(* Logix 5000 project; controller reports 1756-L63 rev 20.15; software revision 20.04; part 44 of 52 *)

        [122].log_data[40].maxminute := 25, [122].log_data[40].valid := 1, [122].log_data[41].min := 0.022540038, [122].log_data[41].max := 0.023128908, [122].log_data[41].total := 82.19256, [122].log_data[41].time := 3600.0, [122].log_data[41].minminute := 6, [122].log_data[41].maxminute := 1, [122].log_data[41].valid := 1, [122].log_data[42].min := 2.2911716, [122].log_data[42].max := 2.2963536, [122].log_data[42].total := 8258.403, [122].log_data[42].time := 3600.0, [122].log_data[42].minminute := 22, [122].log_data[42].maxminute := 41, [122].log_data[42].valid := 1, [122].log_data[43].min := -0.27999878, [122].log_data[43].max := -0.26000214, [122].log_data[43].total := -936.05817, [122].log_data[43].time := 3600.0, [122].log_data[43].minminute := 7, [122].log_data[43].valid := 1, [122].log_data[44].min := -0.30000305, [122].log_data[44].max := -0.27999878, [122].log_data[44].total := -1080.0862, [122].log_data[44].time := 3600.0, [122].log_data[44].maxminute := 20, [122].log_data[44].valid := 1, [122].log_data[45].time := 3600.0, [122].log_data[45].valid := 1, [122].log_data[46].time := 3600.0, [122].log_data[46].valid := 1, [122].log_data[47].time := 3600.0, [122].log_data[47].valid := 1, [122].log_data[48].min := 6.554947, [122].log_data[48].max := 6.9405026, [122].log_data[48].total := 24061.553, [122].log_data[48].time := 3600.0, [122].log_data[48].minminute := 51, [122].log_data[48].maxminute := 30, [122].log_data[48].valid := 1, [122].log_data[49].min := 9.374254, [122].log_data[49].max := 9.504003, [122].log_data[49].total := 34030.01, [122].log_data[49].time := 3600.0, [122].log_data[49].minminute := 59, [122].log_data[49].maxminute := 15, [122].log_data[49].valid := 1, [122].log_data[50].min := 1.5897048, [122].log_data[50].max := 1.6947598, [122].log_data[50].total := 5915.742, [122].log_data[50].time := 3600.0, [122].log_data[50].minminute := 30, [122].log_data[50].maxminute := 37, [122].log_data[50].valid := 1, [122].log_data[51].time := 3600.0, [122].log_data[51].valid := 1, [122].log_data[52].min := -2.959999, [122].log_data[52].max := 0.11999512, [122].log_data[52].total := -7874.2905,
        [122].log_data[52].time := 3600.0, [122].log_data[52].minminute := 54, [122].log_data[52].valid := 1, [122].log_data[53].min := -2.5800018, [122].log_data[53].max := 0.13999939, [122].log_data[53].total := -7446.6367, [122].log_data[53].time := 3600.0, [122].log_data[53].minminute := 9, [122].log_data[53].maxminute := 7, [122].log_data[53].valid := 1, [122].log_data[54].max := 0.5335, [122].log_data[54].total := 1217.6704, [122].log_data[54].time := 3600.0, [122].log_data[54].maxminute := 54, [122].log_data[54].valid := 1, [122].log_data[55].max := 0.5115, [122].log_data[55].total := 1217.3799, [122].log_data[55].time := 3600.0, [122].log_data[55].minminute := 5, [122].log_data[55].maxminute := 7, [122].log_data[55].valid := 1, [122].log_data[56].min := 0.15926416, [122].log_data[56].max := 0.159696, [122].log_data[56].total := 573.94727, [122].log_data[56].time := 3600.0, [122].log_data[56].minminute := 33, [122].log_data[56].maxminute := 2, [122].log_data[56].valid := 1, [122].log_data[57].min := 0.21273394, [122].log_data[57].max := 0.21501088, [122].log_data[57].total := 772.2598, [122].log_data[57].time := 3600.0, [122].log_data[57].minminute := 59, [122].log_data[57].maxminute := 6, [122].log_data[57].valid := 1, [122].log_data[58].time := 3600.0, [122].log_data[58].valid := 1, [122].log_data[59].time := 3600.0, [122].log_data[59].valid := 1, [122].log_data[60].valid := 1, [122].log_data[61].valid := 1, [122].log_data[62].valid := 1, [122].log_data[63].valid := 1, [122].log_data[64].valid := 1, [122].log_data[65].valid := 1, [122].log_data[66].valid := 1, [122].log_data[67].valid := 1, [122].log_data[68].valid := 1, [122].log_data[69].valid := 1, [122].log_data[70].valid := 1, [122].log_data[71].valid := 1, [122].log_data[72].valid := 1, [122].log_data[73].valid := 1, [122].log_data[74].valid := 1, [122].log_data[75].valid := 1, [122].log_data[76].valid := 1, [122].log_data[77].valid := 1, [122].log_data[78].valid := 1, [122].log_data[79].valid := 1, [122].log_data[80].valid := 1,
        [122].log_data[81].valid := 1, [122].log_data[82].valid := 1, [122].log_data[83].valid := 1, [122].log_data[84].valid := 1, [122].log_data[85].valid := 1, [122].log_data[86].valid := 1, [122].log_data[87].valid := 1, [122].log_data[88].valid := 1, [122].log_data[89].valid := 1, [122].log_data[90].valid := 1, [122].log_data[91].valid := 1, [122].log_data[92].valid := 1, [122].log_data[93].valid := 1, [122].log_data[94].valid := 1, [122].log_data[95].valid := 1, [122].log_data[96].valid := 1, [122].log_data[97].valid := 1, [122].log_data[98].valid := 1, [122].log_data[99].valid := 1, [122].log_data[100].valid := 1, [122].log_data[101].valid := 1, [122].log_data[102].valid := 1, [122].log_data[103].valid := 1, [122].log_data[104].valid := 1, [122].log_data[105].valid := 1, [122].log_data[106].valid := 1, [122].log_data[107].valid := 1, [122].log_data[108].valid := 1, [122].log_data[109].valid := 1, [122].log_data[110].valid := 1, [122].log_data[111].valid := 1, [122].log_data[112].valid := 1, [122].log_data[113].valid := 1, [122].log_data[114].valid := 1, [122].log_data[115].valid := 1, [122].log_data[116].valid := 1, [122].log_data[117].valid := 1, [122].log_data[118].valid := 1, [122].log_data[119].valid := 1, [122].log_data[120].valid := 1, [122].log_data[121].valid := 1, [122].log_data[122].valid := 1, [122].log_data[123].valid := 1, [122].log_data[124].valid := 1, [122].time.Year := 2023, [122].time.Month := 1, [122].time.Day := 18, [122].time.Hour := 5, [122].time.Minute := 59, [122].time.Second := 59, [123].log_data[0].min := 1.0, [123].log_data[0].max := 1.0, [123].log_data[0].total := 3600.0, [123].log_data[0].time := 3600.0, [123].log_data[0].valid := 1, [123].log_data[1].time := 3600.0, [123].log_data[1].valid := 1, [123].log_data[2].time := 3600.0, [123].log_data[2].valid := 1, [123].log_data[3].time := 3600.0,
        [123].log_data[3].valid := 1, [123].log_data[4].time := 3600.0, [123].log_data[4].valid := 1, [123].log_data[5].time := 3600.0, [123].log_data[5].valid := 1, [123].log_data[6].time := 3600.0, [123].log_data[6].valid := 1, [123].log_data[7].time := 3600.0, [123].log_data[7].valid := 1, [123].log_data[8].min := 1.0, [123].log_data[8].max := 1.0, [123].log_data[8].total := 3600.0, [123].log_data[8].time := 3600.0, [123].log_data[8].valid := 1, [123].log_data[9].min := 1.0, [123].log_data[9].max := 1.0, [123].log_data[9].total := 3600.0, [123].log_data[9].time := 3600.0, [123].log_data[9].valid := 1, [123].log_data[10].min := 1.0, [123].log_data[10].max := 1.0, [123].log_data[10].total := 3600.0, [123].log_data[10].time := 3600.0, [123].log_data[10].valid := 1, [123].log_data[11].time := 3600.0, [123].log_data[11].valid := 1, [123].log_data[12].min := 1.0, [123].log_data[12].max := 1.0, [123].log_data[12].total := 3600.0, [123].log_data[12].time := 3600.0, [123].log_data[12].valid := 1, [123].log_data[13].min := 1.0, [123].log_data[13].max := 1.0, [123].log_data[13].total := 3600.0, [123].log_data[13].time := 3600.0, [123].log_data[13].valid := 1, [123].log_data[14].time := 3600.0, [123].log_data[14].valid := 1, [123].log_data[15].time := 3600.0, [123].log_data[15].valid := 1, [123].log_data[16].time := 3600.0, [123].log_data[16].valid := 1, [123].log_data[17].min := 1.0, [123].log_data[17].max := 1.0, [123].log_data[17].total := 3600.0, [123].log_data[17].time := 3600.0, [123].log_data[17].valid := 1, [123].log_data[18].time := 3600.0, [123].log_data[18].valid := 1, [123].log_data[19].time := 3600.0, [123].log_data[19].valid := 1, [123].log_data[20].time := 3600.0, [123].log_data[20].valid := 1, [123].log_data[21].min := 1.0, [123].log_data[21].max := 1.0, [123].log_data[21].total := 3600.0, [123].log_data[21].time := 3600.0, [123].log_data[21].valid := 1, [123].log_data[22].time := 3600.0, [123].log_data[22].valid := 1,
        [123].log_data[23].time := 3600.0, [123].log_data[23].valid := 1, [123].log_data[24].time := 3600.0, [123].log_data[24].valid := 1, [123].log_data[25].time := 3600.0, [123].log_data[25].valid := 1, [123].log_data[26].time := 3600.0, [123].log_data[26].valid := 1, [123].log_data[27].time := 3600.0, [123].log_data[27].valid := 1, [123].log_data[28].time := 3600.0, [123].log_data[28].valid := 1, [123].log_data[29].min := 1.0, [123].log_data[29].max := 1.0, [123].log_data[29].total := 3600.0, [123].log_data[29].time := 3600.0, [123].log_data[29].valid := 1, [123].log_data[30].min := 1.0, [123].log_data[30].max := 1.0, [123].log_data[30].total := 3600.0, [123].log_data[30].time := 3600.0, [123].log_data[30].valid := 1, [123].log_data[31].max := 1.0, [123].log_data[31].total := 1440.998, [123].log_data[31].time := 3600.0, [123].log_data[31].minminute := 3, [123].log_data[31].valid := 1, [123].log_data[32].max := 1.0, [123].log_data[32].total := 1630.249, [123].log_data[32].time := 3600.0, [123].log_data[32].maxminute := 4, [123].log_data[32].valid := 1, [123].log_data[33].time := 3600.0, [123].log_data[33].valid := 1, [123].log_data[34].time := 3600.0, [123].log_data[34].valid := 1, [123].log_data[35].max := 1.0, [123].log_data[35].total := 1549.2471, [123].log_data[35].time := 3600.0, [123].log_data[35].maxminute := 10, [123].log_data[35].valid := 1, [123].log_data[36].max := 1.0, [123].log_data[36].total := 1609.498, [123].log_data[36].time := 3600.0, [123].log_data[36].minminute := 8, [123].log_data[36].valid := 1, [123].log_data[37].time := 3600.0, [123].log_data[37].valid := 1, [123].log_data[38].time := 3600.0, [123].log_data[38].valid := 1, [123].log_data[39].min := 0.9947063, [123].log_data[39].max := 1.0056593, [123].log_data[39].total := 3606.119, [123].log_data[39].time := 3600.0, [123].log_data[39].minminute := 20, [123].log_data[39].maxminute := 17, [123].log_data[39].valid := 1, [123].log_data[40].min := 7.602789, [123].log_data[40].max := 7.609111, [123].log_data[40].total := 27387.07,
        [123].log_data[40].time := 3600.0, [123].log_data[40].minminute := 1, [123].log_data[40].valid := 1, [123].log_data[41].min := 0.022540038, [123].log_data[41].max := 0.023128908, [123].log_data[41].total := 82.054955, [123].log_data[41].time := 3600.0, [123].log_data[41].maxminute := 55, [123].log_data[41].valid := 1, [123].log_data[42].min := 2.2912893, [123].log_data[42].max := 2.296118, [123].log_data[42].total := 8258.289, [123].log_data[42].time := 3600.0, [123].log_data[42].minminute := 33, [123].log_data[42].maxminute := 34, [123].log_data[42].valid := 1, [123].log_data[43].min := -0.27999878, [123].log_data[43].max := -0.26000214, [123].log_data[43].total := -936.1481, [123].log_data[43].time := 3600.0, [123].log_data[43].minminute := 14, [123].log_data[43].valid := 1, [123].log_data[44].min := -0.30000305, [123].log_data[44].max := -0.27999878, [123].log_data[44].total := -1080.081, [123].log_data[44].time := 3600.0, [123].log_data[44].valid := 1, [123].log_data[45].time := 3600.0, [123].log_data[45].valid := 1, [123].log_data[46].time := 3600.0, [123].log_data[46].valid := 1, [123].log_data[47].time := 3600.0, [123].log_data[47].valid := 1, [123].log_data[48].min := 6.64371, [123].log_data[48].max := 6.799526, [123].log_data[48].total := 24267.373, [123].log_data[48].time := 3600.0, [123].log_data[48].maxminute := 9, [123].log_data[48].valid := 1, [123].log_data[49].min := 9.362281, [123].log_data[49].max := 9.4512005, [123].log_data[49].total := 33907.27, [123].log_data[49].time := 3600.0, [123].log_data[49].minminute := 5, [123].log_data[49].maxminute := 47, [123].log_data[49].valid := 1, [123].log_data[50].min := 1.5826381, [123].log_data[50].max := 1.6713226, [123].log_data[50].total := 5860.614, [123].log_data[50].time := 3600.0, [123].log_data[50].minminute := 59, [123].log_data[50].valid := 1, [123].log_data[51].time := 3600.0, [123].log_data[51].valid := 1, [123].log_data[52].min := -2.9000015, [123].log_data[52].max := 0.11999512, [123].log_data[52].total := -7866.899, [123].log_data[52].time := 3600.0, [123].log_data[52].minminute := 15, [123].log_data[52].maxminute := 3,
        [123].log_data[52].valid := 1, [123].log_data[53].min := -2.5800018, [123].log_data[53].max := 0.17999268, [123].log_data[53].total := -7646.0073, [123].log_data[53].time := 3600.0, [123].log_data[53].minminute := 54, [123].log_data[53].maxminute := 10, [123].log_data[53].valid := 1, [123].log_data[54].max := 0.535, [123].log_data[54].total := 1217.6685, [123].log_data[54].time := 3600.0, [123].log_data[54].minminute := 3, [123].log_data[54].maxminute := 36, [123].log_data[54].valid := 1, [123].log_data[55].max := 0.522, [123].log_data[55].total := 1254.0444, [123].log_data[55].time := 3600.0, [123].log_data[55].minminute := 8, [123].log_data[55].maxminute := 41, [123].log_data[55].valid := 1, [123].log_data[56].min := 0.15926416, [123].log_data[56].max := 0.15965673, [123].log_data[56].total := 573.912, [123].log_data[56].time := 3600.0, [123].log_data[56].minminute := 38, [123].log_data[56].valid := 1, [123].log_data[57].min := 0.21226284, [123].log_data[57].max := 0.21289097, [123].log_data[57].total := 764.59094, [123].log_data[57].time := 3600.0, [123].log_data[57].minminute := 6, [123].log_data[57].valid := 1, [123].log_data[58].time := 3600.0, [123].log_data[58].valid := 1, [123].log_data[59].time := 3600.0, [123].log_data[59].valid := 1, [123].log_data[60].valid := 1, [123].log_data[61].valid := 1, [123].log_data[62].valid := 1, [123].log_data[63].valid := 1, [123].log_data[64].valid := 1, [123].log_data[65].valid := 1, [123].log_data[66].valid := 1, [123].log_data[67].valid := 1, [123].log_data[68].valid := 1, [123].log_data[69].valid := 1, [123].log_data[70].valid := 1, [123].log_data[71].valid := 1, [123].log_data[72].valid := 1, [123].log_data[73].valid := 1, [123].log_data[74].valid := 1, [123].log_data[75].valid := 1, [123].log_data[76].valid := 1, [123].log_data[77].valid := 1, [123].log_data[78].valid := 1, [123].log_data[79].valid := 1, [123].log_data[80].valid := 1, [123].log_data[81].valid := 1, [123].log_data[82].valid := 1, [123].log_data[83].valid := 1,
        [123].log_data[84].valid := 1, [123].log_data[85].valid := 1, [123].log_data[86].valid := 1, [123].log_data[87].valid := 1, [123].log_data[88].valid := 1, [123].log_data[89].valid := 1, [123].log_data[90].valid := 1, [123].log_data[91].valid := 1, [123].log_data[92].valid := 1, [123].log_data[93].valid := 1, [123].log_data[94].valid := 1, [123].log_data[95].valid := 1, [123].log_data[96].valid := 1, [123].log_data[97].valid := 1, [123].log_data[98].valid := 1, [123].log_data[99].valid := 1, [123].log_data[100].valid := 1, [123].log_data[101].valid := 1, [123].log_data[102].valid := 1, [123].log_data[103].valid := 1, [123].log_data[104].valid := 1, [123].log_data[105].valid := 1, [123].log_data[106].valid := 1, [123].log_data[107].valid := 1, [123].log_data[108].valid := 1, [123].log_data[109].valid := 1, [123].log_data[110].valid := 1, [123].log_data[111].valid := 1, [123].log_data[112].valid := 1, [123].log_data[113].valid := 1, [123].log_data[114].valid := 1, [123].log_data[115].valid := 1, [123].log_data[116].valid := 1, [123].log_data[117].valid := 1, [123].log_data[118].valid := 1, [123].log_data[119].valid := 1, [123].log_data[120].valid := 1, [123].log_data[121].valid := 1, [123].log_data[122].valid := 1, [123].log_data[123].valid := 1, [123].log_data[124].valid := 1, [123].time.Year := 2023, [123].time.Month := 1, [123].time.Day := 18, [123].time.Hour := 6, [123].time.Minute := 59, [123].time.Second := 59, [124].log_data[0].min := 1.0, [124].log_data[0].max := 1.0, [124].log_data[0].total := 3600.0, [124].log_data[0].time := 3600.0, [124].log_data[0].valid := 1, [124].log_data[1].time := 3600.0, [124].log_data[1].valid := 1, [124].log_data[2].time := 3600.0, [124].log_data[2].valid := 1, [124].log_data[3].time := 3600.0, [124].log_data[3].valid := 1, [124].log_data[4].time := 3600.0, [124].log_data[4].valid := 1,
        [124].log_data[5].time := 3600.0, [124].log_data[5].valid := 1, [124].log_data[6].time := 3600.0, [124].log_data[6].valid := 1, [124].log_data[7].time := 3600.0, [124].log_data[7].valid := 1, [124].log_data[8].min := 1.0, [124].log_data[8].max := 1.0, [124].log_data[8].total := 3600.0, [124].log_data[8].time := 3600.0, [124].log_data[8].valid := 1, [124].log_data[9].min := 1.0, [124].log_data[9].max := 1.0, [124].log_data[9].total := 3600.0, [124].log_data[9].time := 3600.0, [124].log_data[9].valid := 1, [124].log_data[10].min := 1.0, [124].log_data[10].max := 1.0, [124].log_data[10].total := 3600.0, [124].log_data[10].time := 3600.0, [124].log_data[10].valid := 1, [124].log_data[11].time := 3600.0, [124].log_data[11].valid := 1, [124].log_data[12].min := 1.0, [124].log_data[12].max := 1.0, [124].log_data[12].total := 3600.0, [124].log_data[12].time := 3600.0, [124].log_data[12].valid := 1, [124].log_data[13].min := 1.0, [124].log_data[13].max := 1.0, [124].log_data[13].total := 3600.0, [124].log_data[13].time := 3600.0, [124].log_data[13].valid := 1, [124].log_data[14].time := 3600.0, [124].log_data[14].valid := 1, [124].log_data[15].time := 3600.0, [124].log_data[15].valid := 1, [124].log_data[16].time := 3600.0, [124].log_data[16].valid := 1, [124].log_data[17].min := 1.0, [124].log_data[17].max := 1.0, [124].log_data[17].total := 3600.0, [124].log_data[17].time := 3600.0, [124].log_data[17].valid := 1, [124].log_data[18].time := 3600.0, [124].log_data[18].valid := 1, [124].log_data[19].time := 3600.0, [124].log_data[19].valid := 1, [124].log_data[20].time := 3600.0, [124].log_data[20].valid := 1, [124].log_data[21].min := 1.0, [124].log_data[21].max := 1.0, [124].log_data[21].total := 3600.0, [124].log_data[21].time := 3600.0, [124].log_data[21].valid := 1, [124].log_data[22].time := 3600.0, [124].log_data[22].valid := 1, [124].log_data[23].time := 3600.0, [124].log_data[23].valid := 1, [124].log_data[24].time := 3600.0,
        [124].log_data[24].valid := 1, [124].log_data[25].time := 3600.0, [124].log_data[25].valid := 1, [124].log_data[26].time := 3600.0, [124].log_data[26].valid := 1, [124].log_data[27].time := 3600.0, [124].log_data[27].valid := 1, [124].log_data[28].time := 3600.0, [124].log_data[28].valid := 1, [124].log_data[29].min := 1.0, [124].log_data[29].max := 1.0, [124].log_data[29].total := 3600.0, [124].log_data[29].time := 3600.0, [124].log_data[29].valid := 1, [124].log_data[30].min := 1.0, [124].log_data[30].max := 1.0, [124].log_data[30].total := 3600.0, [124].log_data[30].time := 3600.0, [124].log_data[30].valid := 1, [124].log_data[31].max := 1.0, [124].log_data[31].total := 1462.998, [124].log_data[31].time := 3600.0, [124].log_data[31].minminute := 6, [124].log_data[31].valid := 1, [124].log_data[32].max := 1.0, [124].log_data[32].total := 1629.998, [124].log_data[32].time := 3600.0, [124].log_data[32].maxminute := 7, [124].log_data[32].valid := 1, [124].log_data[33].time := 3600.0, [124].log_data[33].valid := 1, [124].log_data[34].time := 3600.0, [124].log_data[34].valid := 1, [124].log_data[35].max := 1.0, [124].log_data[35].total := 1440.7471, [124].log_data[35].time := 3600.0, [124].log_data[35].minminute := 1, [124].log_data[35].valid := 1, [124].log_data[36].max := 1.0, [124].log_data[36].total := 1629.7471, [124].log_data[36].time := 3600.0, [124].log_data[36].maxminute := 2, [124].log_data[36].valid := 1, [124].log_data[37].time := 3600.0, [124].log_data[37].valid := 1, [124].log_data[38].time := 3600.0, [124].log_data[38].valid := 1, [124].log_data[39].min := 0.9967084, [124].log_data[39].max := 1.006366, [124].log_data[39].total := 3605.9878, [124].log_data[39].time := 3600.0, [124].log_data[39].minminute := 1, [124].log_data[39].maxminute := 13, [124].log_data[39].valid := 1, [124].log_data[40].min := 7.5928965, [124].log_data[40].max := 7.617629, [124].log_data[40].total := 27379.424, [124].log_data[40].time := 3600.0, [124].log_data[40].minminute := 37, [124].log_data[40].maxminute := 19,
        [124].log_data[40].valid := 1, [124].log_data[41].min := 0.022540038, [124].log_data[41].max := 0.022932617, [124].log_data[41].total := 81.98232, [124].log_data[41].time := 3600.0, [124].log_data[41].valid := 1, [124].log_data[42].min := 2.2910538, [124].log_data[42].max := 2.296236, [124].log_data[42].total := 8258.248, [124].log_data[42].time := 3600.0, [124].log_data[42].minminute := 12, [124].log_data[42].maxminute := 53, [124].log_data[42].valid := 1, [124].log_data[43].min := -0.27999878, [124].log_data[43].max := -0.26000214, [124].log_data[43].total := -936.093, [124].log_data[43].time := 3600.0, [124].log_data[43].valid := 1, [124].log_data[44].min := -0.30000305, [124].log_data[44].max := -0.27999878, [124].log_data[44].total := -1080.081, [124].log_data[44].time := 3600.0, [124].log_data[44].maxminute := 29, [124].log_data[44].valid := 1, [124].log_data[45].time := 3600.0, [124].log_data[45].valid := 1, [124].log_data[46].time := 3600.0, [124].log_data[46].valid := 1, [124].log_data[47].time := 3600.0, [124].log_data[47].valid := 1, [124].log_data[48].min := 6.598092, [124].log_data[48].max := 6.695649, [124].log_data[48].total := 23905.256, [124].log_data[48].time := 3600.0, [124].log_data[48].minminute := 32, [124].log_data[48].valid := 1, [124].log_data[49].min := 9.315563, [124].log_data[49].max := 9.46926, [124].log_data[49].total := 33868.32, [124].log_data[49].time := 3600.0, [124].log_data[49].minminute := 59, [124].log_data[49].maxminute := 11, [124].log_data[49].valid := 1, [124].log_data[50].min := 1.487005, [124].log_data[50].max := 1.5914714, [124].log_data[50].total := 5555.008, [124].log_data[50].time := 3600.0, [124].log_data[50].minminute := 59, [124].log_data[50].valid := 1, [124].log_data[51].time := 3600.0, [124].log_data[51].valid := 1, [124].log_data[52].min := -3.040001, [124].log_data[52].max := 0.11999512, [124].log_data[52].total := -7958.977, [124].log_data[52].time := 3600.0, [124].log_data[52].minminute := 39, [124].log_data[52].maxminute := 6, [124].log_data[52].valid := 1, [124].log_data[53].min := -2.6600037, [124].log_data[53].max := 0.22000122,
        [124].log_data[53].total := -7429.467, [124].log_data[53].time := 3600.0, [124].log_data[53].minminute := 2, [124].log_data[53].maxminute := 23, [124].log_data[53].valid := 1, [124].log_data[54].max := 0.551, [124].log_data[54].total := 1228.46, [124].log_data[54].time := 3600.0, [124].log_data[54].minminute := 6, [124].log_data[54].maxminute := 39, [124].log_data[54].valid := 1, [124].log_data[55].max := 0.5345, [124].log_data[55].total := 1217.3112, [124].log_data[55].time := 3600.0, [124].log_data[55].minminute := 1, [124].log_data[55].maxminute := 2, [124].log_data[55].valid := 1, [124].log_data[56].min := 0.1592249, [124].log_data[56].max := 0.15965673, [124].log_data[56].total := 573.8516, [124].log_data[56].time := 3600.0, [124].log_data[56].maxminute := 25, [124].log_data[56].valid := 1, [124].log_data[57].min := 0.20849404, [124].log_data[57].max := 0.21261616, [124].log_data[57].total := 761.44434, [124].log_data[57].time := 3600.0, [124].log_data[57].minminute := 59, [124].log_data[57].maxminute := 3, [124].log_data[57].valid := 1, [124].log_data[58].time := 3600.0, [124].log_data[58].valid := 1, [124].log_data[59].time := 3600.0, [124].log_data[59].valid := 1, [124].log_data[60].valid := 1, [124].log_data[61].valid := 1, [124].log_data[62].valid := 1, [124].log_data[63].valid := 1, [124].log_data[64].valid := 1, [124].log_data[65].valid := 1, [124].log_data[66].valid := 1, [124].log_data[67].valid := 1, [124].log_data[68].valid := 1, [124].log_data[69].valid := 1, [124].log_data[70].valid := 1, [124].log_data[71].valid := 1, [124].log_data[72].valid := 1, [124].log_data[73].valid := 1, [124].log_data[74].valid := 1, [124].log_data[75].valid := 1, [124].log_data[76].valid := 1, [124].log_data[77].valid := 1, [124].log_data[78].valid := 1, [124].log_data[79].valid := 1, [124].log_data[80].valid := 1, [124].log_data[81].valid := 1, [124].log_data[82].valid := 1, [124].log_data[83].valid := 1, [124].log_data[84].valid := 1, [124].log_data[85].valid := 1,
        [124].log_data[86].valid := 1, [124].log_data[87].valid := 1, [124].log_data[88].valid := 1, [124].log_data[89].valid := 1, [124].log_data[90].valid := 1, [124].log_data[91].valid := 1, [124].log_data[92].valid := 1, [124].log_data[93].valid := 1, [124].log_data[94].valid := 1, [124].log_data[95].valid := 1, [124].log_data[96].valid := 1, [124].log_data[97].valid := 1, [124].log_data[98].valid := 1, [124].log_data[99].valid := 1, [124].log_data[100].valid := 1, [124].log_data[101].valid := 1, [124].log_data[102].valid := 1, [124].log_data[103].valid := 1, [124].log_data[104].valid := 1, [124].log_data[105].valid := 1, [124].log_data[106].valid := 1, [124].log_data[107].valid := 1, [124].log_data[108].valid := 1, [124].log_data[109].valid := 1, [124].log_data[110].valid := 1, [124].log_data[111].valid := 1, [124].log_data[112].valid := 1, [124].log_data[113].valid := 1, [124].log_data[114].valid := 1, [124].log_data[115].valid := 1, [124].log_data[116].valid := 1, [124].log_data[117].valid := 1, [124].log_data[118].valid := 1, [124].log_data[119].valid := 1, [124].log_data[120].valid := 1, [124].log_data[121].valid := 1, [124].log_data[122].valid := 1, [124].log_data[123].valid := 1, [124].log_data[124].valid := 1, [124].time.Year := 2023, [124].time.Month := 1, [124].time.Day := 18, [124].time.Hour := 7, [124].time.Minute := 59, [124].time.Second := 59, [125].log_data[0].min := 1.0, [125].log_data[0].max := 1.0, [125].log_data[0].total := 3599.5, [125].log_data[0].time := 3599.5, [125].log_data[0].valid := 1, [125].log_data[1].max := 1.0, [125].log_data[1].total := 535.0, [125].log_data[1].time := 3599.5, [125].log_data[1].maxminute := 45, [125].log_data[1].valid := 1, [125].log_data[2].max := 1.0, [125].log_data[2].total := 531.5, [125].log_data[2].time := 3599.5, [125].log_data[2].maxminute := 45, [125].log_data[2].valid := 1,
        [125].log_data[3].time := 3599.5, [125].log_data[3].valid := 1, [125].log_data[4].time := 3599.5, [125].log_data[4].valid := 1, [125].log_data[5].max := 1.0, [125].log_data[5].total := 240.0, [125].log_data[5].time := 3599.5, [125].log_data[5].maxminute := 47, [125].log_data[5].valid := 1, [125].log_data[6].time := 3599.5, [125].log_data[6].valid := 1, [125].log_data[7].time := 3599.5, [125].log_data[7].valid := 1, [125].log_data[8].min := 1.0, [125].log_data[8].max := 1.0, [125].log_data[8].total := 3599.5, [125].log_data[8].time := 3599.5, [125].log_data[8].valid := 1, [125].log_data[9].min := 1.0, [125].log_data[9].max := 1.0, [125].log_data[9].total := 3599.5, [125].log_data[9].time := 3599.5, [125].log_data[9].valid := 1, [125].log_data[10].min := 1.0, [125].log_data[10].max := 1.0, [125].log_data[10].total := 3599.5, [125].log_data[10].time := 3599.5, [125].log_data[10].valid := 1, [125].log_data[11].time := 3599.5, [125].log_data[11].valid := 1, [125].log_data[12].min := 1.0, [125].log_data[12].max := 1.0, [125].log_data[12].total := 3599.5, [125].log_data[12].time := 3599.5, [125].log_data[12].valid := 1, [125].log_data[13].min := 1.0, [125].log_data[13].max := 1.0, [125].log_data[13].total := 3599.5, [125].log_data[13].time := 3599.5, [125].log_data[13].valid := 1, [125].log_data[14].time := 3599.5, [125].log_data[14].valid := 1, [125].log_data[15].time := 3599.5, [125].log_data[15].valid := 1, [125].log_data[16].max := 1.0, [125].log_data[16].total := 7.5, [125].log_data[16].time := 3599.5, [125].log_data[16].maxminute := 30, [125].log_data[16].valid := 1, [125].log_data[17].max := 1.0, [125].log_data[17].total := 918.249, [125].log_data[17].time := 3599.5, [125].log_data[17].minminute := 2, [125].log_data[17].valid := 1, [125].log_data[18].time := 3599.5, [125].log_data[18].valid := 1, [125].log_data[19].time := 3599.5, [125].log_data[19].valid := 1, [125].log_data[20].time := 3599.5, [125].log_data[20].valid := 1,
        [125].log_data[21].min := 1.0, [125].log_data[21].max := 1.0, [125].log_data[21].total := 3599.5, [125].log_data[21].time := 3599.5, [125].log_data[21].valid := 1, [125].log_data[22].time := 3599.5, [125].log_data[22].valid := 1, [125].log_data[23].time := 3599.5, [125].log_data[23].valid := 1, [125].log_data[24].time := 3599.5, [125].log_data[24].valid := 1, [125].log_data[25].time := 3599.5, [125].log_data[25].valid := 1, [125].log_data[26].time := 3599.5, [125].log_data[26].valid := 1, [125].log_data[27].time := 3599.5, [125].log_data[27].valid := 1, [125].log_data[28].time := 3599.5, [125].log_data[28].valid := 1, [125].log_data[29].min := 1.0, [125].log_data[29].max := 1.0, [125].log_data[29].total := 3599.5, [125].log_data[29].time := 3599.5, [125].log_data[29].valid := 1, [125].log_data[30].min := 1.0, [125].log_data[30].max := 1.0, [125].log_data[30].total := 3599.5, [125].log_data[30].time := 3599.5, [125].log_data[30].valid := 1, [125].log_data[31].max := 1.0, [125].log_data[31].total := 1629.998, [125].log_data[31].time := 3599.5, [125].log_data[31].valid := 1, [125].log_data[32].max := 1.0, [125].log_data[32].total := 1506.2471, [125].log_data[32].time := 3599.5, [125].log_data[32].maxminute := 10, [125].log_data[32].valid := 1, [125].log_data[33].time := 3599.5, [125].log_data[33].valid := 1, [125].log_data[34].time := 3599.5, [125].log_data[34].valid := 1, [125].log_data[35].max := 1.0, [125].log_data[35].total := 1440.2471, [125].log_data[35].time := 3599.5, [125].log_data[35].minminute := 4, [125].log_data[35].valid := 1, [125].log_data[36].max := 1.0, [125].log_data[36].total := 1629.7471, [125].log_data[36].time := 3599.5, [125].log_data[36].maxminute := 5, [125].log_data[36].valid := 1, [125].log_data[37].max := 7.6321344, [125].log_data[37].total := 3523.888, [125].log_data[37].time := 3599.5, [125].log_data[37].maxminute := 45, [125].log_data[37].valid := 1, [125].log_data[38].time := 3599.5, [125].log_data[38].valid := 1, [125].log_data[39].min := 0.9961195,
        [125].log_data[39].max := 1.0217944, [125].log_data[39].total := 3610.299, [125].log_data[39].time := 3599.5, [125].log_data[39].minminute := 37, [125].log_data[39].maxminute := 52, [125].log_data[39].valid := 1, [125].log_data[40].min := 7.5854764, [125].log_data[40].max := 7.617629, [125].log_data[40].total := 27378.451, [125].log_data[40].time := 3599.5, [125].log_data[40].minminute := 33, [125].log_data[40].maxminute := 37, [125].log_data[40].valid := 1, [125].log_data[41].min := 0.022540038, [125].log_data[41].max := 0.023128908, [125].log_data[41].total := 82.010216, [125].log_data[41].time := 3599.5, [125].log_data[41].maxminute := 20, [125].log_data[41].valid := 1, [125].log_data[42].min := 2.291525, [125].log_data[42].max := 2.2960005, [125].log_data[42].total := 8257.242, [125].log_data[42].time := 3599.5, [125].log_data[42].minminute := 4, [125].log_data[42].maxminute := 10, [125].log_data[42].valid := 1, [125].log_data[43].min := -0.27999878, [125].log_data[43].max := -0.26000214, [125].log_data[43].total := -959.55176, [125].log_data[43].time := 3599.5, [125].log_data[43].minminute := 2, [125].log_data[43].valid := 1, [125].log_data[44].min := -0.3199997, [125].log_data[44].max := -0.27999878, [125].log_data[44].total := -1093.7062, [125].log_data[44].time := 3599.5, [125].log_data[44].minminute := 41, [125].log_data[44].maxminute := 14, [125].log_data[44].valid := 1, [125].log_data[45].time := 3599.5, [125].log_data[45].valid := 1, [125].log_data[46].time := 3599.5, [125].log_data[46].valid := 1, [125].log_data[47].time := 3599.5, [125].log_data[47].valid := 1, [125].log_data[48].min := 6.6110077, [125].log_data[48].max := 7.693476, [125].log_data[48].total := 24599.236, [125].log_data[48].time := 3599.5, [125].log_data[48].maxminute := 52, [125].log_data[48].valid := 1, [125].log_data[49].min := 9.285924, [125].log_data[49].max := 9.409587, [125].log_data[49].total := 33653.25, [125].log_data[49].time := 3599.5, [125].log_data[49].minminute := 13, [125].log_data[49].maxminute := 58, [125].log_data[49].valid := 1, [125].log_data[50].min := 1.4267042, [125].log_data[50].max := 1.5370593,
        [125].log_data[50].total := 5289.228, [125].log_data[50].time := 3599.5, [125].log_data[50].minminute := 47, [125].log_data[50].maxminute := 54, [125].log_data[50].valid := 1, [125].log_data[51].time := 3599.5, [125].log_data[51].valid := 1, [125].log_data[52].min := -2.8600006, [125].log_data[52].max := 0.11999512, [125].log_data[52].total := -8118.5156, [125].log_data[52].time := 3599.5, [125].log_data[52].minminute := 45, [125].log_data[52].valid := 1, [125].log_data[53].min := -2.600006, [125].log_data[53].max := 0.16000366, [125].log_data[53].total := -7416.408, [125].log_data[53].time := 3599.5, [125].log_data[53].minminute := 56, [125].log_data[53].maxminute := 5, [125].log_data[53].valid := 1, [125].log_data[54].max := 0.52099997, [125].log_data[54].total := 1243.1195, [125].log_data[54].time := 3599.5, [125].log_data[54].maxminute := 42, [125].log_data[54].valid := 1, [125].log_data[55].max := 0.5385, [125].log_data[55].total := 1216.6307, [125].log_data[55].time := 3599.5, [125].log_data[55].minminute := 4, [125].log_data[55].maxminute := 16, [125].log_data[55].valid := 1, [125].log_data[56].min := 0.1592249, [125].log_data[56].max := 0.15961748, [125].log_data[56].total := 573.72363, [125].log_data[56].time := 3599.5, [125].log_data[56].minminute := 44, [125].log_data[56].valid := 1, [125].log_data[57].min := 0.20079942, [125].log_data[57].max := 0.20869033, [125].log_data[57].total := 733.58307, [125].log_data[57].time := 3599.5, [125].log_data[57].minminute := 54, [125].log_data[57].valid := 1, [125].log_data[58].time := 3599.5, [125].log_data[58].valid := 1, [125].log_data[59].time := 3599.5, [125].log_data[59].valid := 1, [125].log_data[60].valid := 1, [125].log_data[61].valid := 1, [125].log_data[62].valid := 1, [125].log_data[63].valid := 1, [125].log_data[64].valid := 1, [125].log_data[65].valid := 1, [125].log_data[66].valid := 1, [125].log_data[67].valid := 1, [125].log_data[68].valid := 1, [125].log_data[69].valid := 1, [125].log_data[70].valid := 1, [125].log_data[71].valid := 1, [125].log_data[72].valid := 1,
        [125].log_data[73].valid := 1, [125].log_data[74].valid := 1, [125].log_data[75].valid := 1, [125].log_data[76].valid := 1, [125].log_data[77].valid := 1, [125].log_data[78].valid := 1, [125].log_data[79].valid := 1, [125].log_data[80].valid := 1, [125].log_data[81].valid := 1, [125].log_data[82].valid := 1, [125].log_data[83].valid := 1, [125].log_data[84].valid := 1, [125].log_data[85].valid := 1, [125].log_data[86].valid := 1, [125].log_data[87].valid := 1, [125].log_data[88].valid := 1, [125].log_data[89].valid := 1, [125].log_data[90].valid := 1, [125].log_data[91].valid := 1, [125].log_data[92].valid := 1, [125].log_data[93].valid := 1, [125].log_data[94].valid := 1, [125].log_data[95].valid := 1, [125].log_data[96].valid := 1, [125].log_data[97].valid := 1, [125].log_data[98].valid := 1, [125].log_data[99].valid := 1, [125].log_data[100].valid := 1, [125].log_data[101].valid := 1, [125].log_data[102].valid := 1, [125].log_data[103].valid := 1, [125].log_data[104].valid := 1, [125].log_data[105].valid := 1, [125].log_data[106].valid := 1, [125].log_data[107].valid := 1, [125].log_data[108].valid := 1, [125].log_data[109].valid := 1, [125].log_data[110].valid := 1, [125].log_data[111].valid := 1, [125].log_data[112].valid := 1, [125].log_data[113].valid := 1, [125].log_data[114].valid := 1, [125].log_data[115].valid := 1, [125].log_data[116].valid := 1, [125].log_data[117].valid := 1, [125].log_data[118].valid := 1, [125].log_data[119].valid := 1, [125].log_data[120].valid := 1, [125].log_data[121].valid := 1, [125].log_data[122].valid := 1, [125].log_data[123].valid := 1, [125].log_data[124].valid := 1, [125].time.Year := 2023, [125].time.Month := 1, [125].time.Day := 18, [125].time.Hour := 8, [125].time.Minute := 59, [125].time.Second := 59, [126].log_data[0].min := 1.0, [126].log_data[0].max := 1.0,
        [126].log_data[0].total := 3600.0, [126].log_data[0].time := 3600.0, [126].log_data[0].valid := 1, [126].log_data[1].max := 1.0, [126].log_data[1].total := 168.5, [126].log_data[1].time := 3600.0, [126].log_data[1].maxminute := 43, [126].log_data[1].valid := 1, [126].log_data[2].max := 1.0, [126].log_data[2].total := 165.0, [126].log_data[2].time := 3600.0, [126].log_data[2].maxminute := 44, [126].log_data[2].valid := 1, [126].log_data[3].time := 3600.0, [126].log_data[3].valid := 1, [126].log_data[4].time := 3600.0, [126].log_data[4].valid := 1, [126].log_data[5].time := 3600.0, [126].log_data[5].valid := 1, [126].log_data[6].time := 3600.0, [126].log_data[6].valid := 1, [126].log_data[7].time := 3600.0, [126].log_data[7].valid := 1, [126].log_data[8].max := 1.0, [126].log_data[8].total := 1325.251, [126].log_data[8].time := 3600.0, [126].log_data[8].minminute := 22, [126].log_data[8].valid := 1, [126].log_data[9].max := 1.0, [126].log_data[9].total := 1328.251, [126].log_data[9].time := 3600.0, [126].log_data[9].minminute := 22, [126].log_data[9].valid := 1, [126].log_data[10].min := 1.0, [126].log_data[10].max := 1.0, [126].log_data[10].total := 3600.0, [126].log_data[10].time := 3600.0, [126].log_data[10].valid := 1, [126].log_data[11].time := 3600.0, [126].log_data[11].valid := 1, [126].log_data[12].min := 1.0, [126].log_data[12].max := 1.0, [126].log_data[12].total := 3600.0, [126].log_data[12].time := 3600.0, [126].log_data[12].valid := 1, [126].log_data[13].min := 1.0, [126].log_data[13].max := 1.0, [126].log_data[13].total := 3600.0, [126].log_data[13].time := 3600.0, [126].log_data[13].valid := 1, [126].log_data[14].time := 3600.0, [126].log_data[14].valid := 1, [126].log_data[15].time := 3600.0, [126].log_data[15].valid := 1, [126].log_data[16].time := 3600.0, [126].log_data[16].valid := 1, [126].log_data[17].min := 1.0, [126].log_data[17].max := 1.0, [126].log_data[17].total := 3600.0, [126].log_data[17].time := 3600.0,
        [126].log_data[17].valid := 1, [126].log_data[18].time := 3600.0, [126].log_data[18].valid := 1, [126].log_data[19].time := 3600.0, [126].log_data[19].valid := 1, [126].log_data[20].time := 3600.0, [126].log_data[20].valid := 1, [126].log_data[21].min := 1.0, [126].log_data[21].max := 1.0, [126].log_data[21].total := 3600.0, [126].log_data[21].time := 3600.0, [126].log_data[21].valid := 1, [126].log_data[22].time := 3600.0, [126].log_data[22].valid := 1, [126].log_data[23].time := 3600.0, [126].log_data[23].valid := 1, [126].log_data[24].time := 3600.0, [126].log_data[24].valid := 1, [126].log_data[25].time := 3600.0, [126].log_data[25].valid := 1, [126].log_data[26].time := 3600.0, [126].log_data[26].valid := 1, [126].log_data[27].time := 3600.0, [126].log_data[27].valid := 1, [126].log_data[28].time := 3600.0, [126].log_data[28].valid := 1, [126].log_data[29].min := 1.0, [126].log_data[29].max := 1.0, [126].log_data[29].total := 3600.0, [126].log_data[29].time := 3600.0, [126].log_data[29].valid := 1, [126].log_data[30].min := 1.0, [126].log_data[30].max := 1.0, [126].log_data[30].total := 3600.0, [126].log_data[30].time := 3600.0, [126].log_data[30].valid := 1, [126].log_data[31].max := 1.0, [126].log_data[31].total := 543.249, [126].log_data[31].time := 3600.0, [126].log_data[31].maxminute := 3, [126].log_data[31].valid := 1, [126].log_data[32].max := 1.0, [126].log_data[32].total := 609.249, [126].log_data[32].time := 3600.0, [126].log_data[32].minminute := 2, [126].log_data[32].valid := 1, [126].log_data[33].time := 3600.0, [126].log_data[33].valid := 1, [126].log_data[34].time := 3600.0, [126].log_data[34].valid := 1, [126].log_data[35].max := 1.0, [126].log_data[35].total := 612.249, [126].log_data[35].time := 3600.0, [126].log_data[35].minminute := 7, [126].log_data[35].valid := 1, [126].log_data[36].max := 1.0, [126].log_data[36].total := 543.249, [126].log_data[36].time := 3600.0, [126].log_data[36].maxminute := 9, [126].log_data[36].valid := 1,
        [126].log_data[37].max := 7.0464015, [126].log_data[37].total := 737.99945, [126].log_data[37].time := 3600.0, [126].log_data[37].maxminute := 44, [126].log_data[37].valid := 1, [126].log_data[38].time := 3600.0, [126].log_data[38].valid := 1, [126].log_data[39].min := 0.99541295, [126].log_data[39].max := 1.0167301, [126].log_data[39].total := 3613.6487, [126].log_data[39].time := 3600.0, [126].log_data[39].minminute := 16, [126].log_data[39].maxminute := 50, [126].log_data[39].valid := 1, [126].log_data[40].min := 7.585752, [126].log_data[40].max := 7.6244993, [126].log_data[40].total := 27383.654, [126].log_data[40].time := 3600.0, [126].log_data[40].minminute := 41, [126].log_data[40].maxminute := 47, [126].log_data[40].valid := 1, [126].log_data[41].min := 0.022540038, [126].log_data[41].max := 0.023128908, [126].log_data[41].total := 82.20095, [126].log_data[41].time := 3600.0, [126].log_data[41].minminute := 1, [126].log_data[41].maxminute := 11, [126].log_data[41].valid := 1, [126].log_data[42].min := 2.2910538, [126].log_data[42].max := 2.296118, [126].log_data[42].total := 8258.457, [126].log_data[42].time := 3600.0, [126].log_data[42].minminute := 20, [126].log_data[42].maxminute := 43, [126].log_data[42].valid := 1, [126].log_data[43].min := -0.27999878, [126].log_data[43].max := -0.23999786, [126].log_data[43].total := -941.8486, [126].log_data[43].time := 3600.0, [126].log_data[43].maxminute := 40, [126].log_data[43].valid := 1, [126].log_data[44].min := -0.3199997, [126].log_data[44].max := -0.27999878, [126].log_data[44].total := -1068.5466, [126].log_data[44].time := 3600.0, [126].log_data[44].maxminute := 29, [126].log_data[44].valid := 1, [126].log_data[45].time := 3600.0, [126].log_data[45].valid := 1, [126].log_data[46].time := 3600.0, [126].log_data[46].valid := 1, [126].log_data[47].time := 3600.0, [126].log_data[47].valid := 1, [126].log_data[48].min := 7.196898, [126].log_data[48].max := 7.622027, [126].log_data[48].total := 26487.303, [126].log_data[48].time := 3600.0, [126].log_data[48].minminute := 32, [126].log_data[48].valid := 1, [126].log_data[49].min := 9.278858,
        [126].log_data[49].max := 9.396239, [126].log_data[49].total := 33586.234, [126].log_data[49].time := 3600.0, [126].log_data[49].minminute := 25, [126].log_data[49].valid := 1, [126].log_data[50].min := 1.4989002, [126].log_data[50].max := 1.6101975, [126].log_data[50].total := 5649.5786, [126].log_data[50].time := 3600.0, [126].log_data[50].minminute := 21, [126].log_data[50].maxminute := 58, [126].log_data[50].valid := 1, [126].log_data[51].time := 3600.0, [126].log_data[51].valid := 1, [126].log_data[52].min := -2.959999, [126].log_data[52].max := 0.1000061, [126].log_data[52].total := -6199.621, [126].log_data[52].time := 3600.0, [126].log_data[52].minminute := 3, [126].log_data[52].maxminute := 2, [126].log_data[52].valid := 1, [126].log_data[53].min := -2.6200027, [126].log_data[53].max := 0.11999512, [126].log_data[53].total := -5728.463, [126].log_data[53].time := 3600.0, [126].log_data[53].minminute := 11, [126].log_data[53].maxminute := 8, [126].log_data[53].valid := 1, [126].log_data[54].max := 0.5375, [126].log_data[54].total := 457.70105, [126].log_data[54].time := 3600.0, [126].log_data[54].minminute := 2, [126].log_data[54].maxminute := 3, [126].log_data[54].valid := 1, [126].log_data[55].max := 0.5195, [126].log_data[55].total := 458.91534, [126].log_data[55].time := 3600.0, [126].log_data[55].minminute := 7, [126].log_data[55].maxminute := 9, [126].log_data[55].valid := 1, [126].log_data[56].min := 0.15918565, [126].log_data[56].max := 0.15973525, [126].log_data[56].total := 573.97205, [126].log_data[56].time := 3600.0, [126].log_data[56].minminute := 2, [126].log_data[56].maxminute := 56, [126].log_data[56].valid := 1, [126].log_data[57].min := 0.20068164, [126].log_data[57].max := 0.20111348, [126].log_data[57].total := 723.1268, [126].log_data[57].time := 3600.0, [126].log_data[57].minminute := 11, [126].log_data[57].maxminute := 47, [126].log_data[57].valid := 1, [126].log_data[58].time := 3600.0, [126].log_data[58].valid := 1, [126].log_data[59].time := 3600.0, [126].log_data[59].valid := 1, [126].log_data[60].valid := 1, [126].log_data[61].valid := 1,
        [126].log_data[62].valid := 1, [126].log_data[63].valid := 1, [126].log_data[64].valid := 1, [126].log_data[65].valid := 1, [126].log_data[66].valid := 1, [126].log_data[67].valid := 1, [126].log_data[68].valid := 1, [126].log_data[69].valid := 1, [126].log_data[70].valid := 1, [126].log_data[71].valid := 1, [126].log_data[72].valid := 1, [126].log_data[73].valid := 1, [126].log_data[74].valid := 1, [126].log_data[75].valid := 1, [126].log_data[76].valid := 1, [126].log_data[77].valid := 1, [126].log_data[78].valid := 1, [126].log_data[79].valid := 1, [126].log_data[80].valid := 1, [126].log_data[81].valid := 1, [126].log_data[82].valid := 1, [126].log_data[83].valid := 1, [126].log_data[84].valid := 1, [126].log_data[85].valid := 1, [126].log_data[86].valid := 1, [126].log_data[87].valid := 1, [126].log_data[88].valid := 1, [126].log_data[89].valid := 1, [126].log_data[90].valid := 1, [126].log_data[91].valid := 1, [126].log_data[92].valid := 1, [126].log_data[93].valid := 1, [126].log_data[94].valid := 1, [126].log_data[95].valid := 1, [126].log_data[96].valid := 1, [126].log_data[97].valid := 1, [126].log_data[98].valid := 1, [126].log_data[99].valid := 1, [126].log_data[100].valid := 1, [126].log_data[101].valid := 1, [126].log_data[102].valid := 1, [126].log_data[103].valid := 1, [126].log_data[104].valid := 1, [126].log_data[105].valid := 1, [126].log_data[106].valid := 1, [126].log_data[107].valid := 1, [126].log_data[108].valid := 1, [126].log_data[109].valid := 1, [126].log_data[110].valid := 1, [126].log_data[111].valid := 1, [126].log_data[112].valid := 1, [126].log_data[113].valid := 1, [126].log_data[114].valid := 1, [126].log_data[115].valid := 1, [126].log_data[116].valid := 1, [126].log_data[117].valid := 1, [126].log_data[118].valid := 1, [126].log_data[119].valid := 1, [126].log_data[120].valid := 1, [126].log_data[121].valid := 1,
        [126].log_data[122].valid := 1, [126].log_data[123].valid := 1, [126].log_data[124].valid := 1, [126].time.Year := 2023, [126].time.Month := 1, [126].time.Day := 18, [126].time.Hour := 9, [126].time.Minute := 59, [126].time.Second := 59, [127].log_data[0].min := 1.0, [127].log_data[0].max := 1.0, [127].log_data[0].total := 3600.0, [127].log_data[0].time := 3600.0, [127].log_data[0].valid := 1, [127].log_data[1].time := 3600.0, [127].log_data[1].valid := 1, [127].log_data[2].time := 3600.0, [127].log_data[2].valid := 1, [127].log_data[3].time := 3600.0, [127].log_data[3].valid := 1, [127].log_data[4].time := 3600.0, [127].log_data[4].valid := 1, [127].log_data[5].time := 3600.0, [127].log_data[5].valid := 1, [127].log_data[6].time := 3600.0, [127].log_data[6].valid := 1, [127].log_data[7].time := 3600.0, [127].log_data[7].valid := 1, [127].log_data[8].time := 3600.0, [127].log_data[8].valid := 1, [127].log_data[9].time := 3600.0, [127].log_data[9].valid := 1, [127].log_data[10].min := 1.0, [127].log_data[10].max := 1.0, [127].log_data[10].total := 3600.0, [127].log_data[10].time := 3600.0, [127].log_data[10].valid := 1, [127].log_data[11].time := 3600.0, [127].log_data[11].valid := 1, [127].log_data[12].min := 1.0, [127].log_data[12].max := 1.0, [127].log_data[12].total := 3600.0, [127].log_data[12].time := 3600.0, [127].log_data[12].valid := 1, [127].log_data[13].min := 1.0, [127].log_data[13].max := 1.0, [127].log_data[13].total := 3600.0, [127].log_data[13].time := 3600.0, [127].log_data[13].valid := 1, [127].log_data[14].time := 3600.0, [127].log_data[14].valid := 1, [127].log_data[15].time := 3600.0, [127].log_data[15].valid := 1, [127].log_data[16].time := 3600.0, [127].log_data[16].valid := 1, [127].log_data[17].min := 1.0, [127].log_data[17].max := 1.0, [127].log_data[17].total := 3600.0, [127].log_data[17].time := 3600.0, [127].log_data[17].valid := 1,
        [127].log_data[18].time := 3600.0, [127].log_data[18].valid := 1, [127].log_data[19].time := 3600.0, [127].log_data[19].valid := 1, [127].log_data[20].time := 3600.0, [127].log_data[20].valid := 1, [127].log_data[21].min := 1.0, [127].log_data[21].max := 1.0, [127].log_data[21].total := 3600.0, [127].log_data[21].time := 3600.0, [127].log_data[21].valid := 1, [127].log_data[22].time := 3600.0, [127].log_data[22].valid := 1, [127].log_data[23].time := 3600.0, [127].log_data[23].valid := 1, [127].log_data[24].time := 3600.0, [127].log_data[24].valid := 1, [127].log_data[25].time := 3600.0, [127].log_data[25].valid := 1, [127].log_data[26].time := 3600.0, [127].log_data[26].valid := 1, [127].log_data[27].time := 3600.0, [127].log_data[27].valid := 1, [127].log_data[28].time := 3600.0, [127].log_data[28].valid := 1, [127].log_data[29].min := 1.0, [127].log_data[29].max := 1.0, [127].log_data[29].total := 3600.0, [127].log_data[29].time := 3600.0, [127].log_data[29].valid := 1, [127].log_data[30].min := 1.0, [127].log_data[30].max := 1.0, [127].log_data[30].total := 3600.0, [127].log_data[30].time := 3600.0, [127].log_data[30].valid := 1, [127].log_data[31].time := 3600.0, [127].log_data[31].valid := 1, [127].log_data[32].time := 3600.0, [127].log_data[32].valid := 1, [127].log_data[33].time := 3600.0, [127].log_data[33].valid := 1, [127].log_data[34].time := 3600.0, [127].log_data[34].valid := 1, [127].log_data[35].time := 3600.0, [127].log_data[35].valid := 1, [127].log_data[36].time := 3600.0, [127].log_data[36].valid := 1, [127].log_data[37].time := 3600.0, [127].log_data[37].valid := 1, [127].log_data[38].time := 3600.0, [127].log_data[38].valid := 1, [127].log_data[39].min := 1.008957, [127].log_data[39].max := 1.0176724, [127].log_data[39].total := 3649.0654, [127].log_data[39].time := 3600.0, [127].log_data[39].minminute := 13, [127].log_data[39].maxminute := 16, [127].log_data[39].valid := 1, [127].log_data[40].min := 7.5885, [127].log_data[40].max := 7.615981,
        [127].log_data[40].total := 27383.064, [127].log_data[40].time := 3600.0, [127].log_data[40].minminute := 5, [127].log_data[40].maxminute := 22, [127].log_data[40].valid := 1, [127].log_data[41].min := 0.022540038, [127].log_data[41].max := 0.022932617, [127].log_data[41].total := 81.807915, [127].log_data[41].time := 3600.0, [127].log_data[41].minminute := 1, [127].log_data[41].valid := 1, [127].log_data[42].min := 2.2912893, [127].log_data[42].max := 2.296236, [127].log_data[42].total := 8258.101, [127].log_data[42].time := 3600.0, [127].log_data[42].minminute := 11, [127].log_data[42].maxminute := 46, [127].log_data[42].valid := 1, [127].log_data[43].min := -0.26000214, [127].log_data[43].max := -0.23999786, [127].log_data[43].total := -898.9608, [127].log_data[43].time := 3600.0, [127].log_data[43].valid := 1, [127].log_data[44].min := -0.30000305, [127].log_data[44].max := -0.27999878, [127].log_data[44].total := -1007.90155, [127].log_data[44].time := 3600.0, [127].log_data[44].minminute := 56, [127].log_data[44].valid := 1, [127].log_data[45].time := 3600.0, [127].log_data[45].valid := 1, [127].log_data[46].time := 3600.0, [127].log_data[46].valid := 1, [127].log_data[47].time := 3600.0, [127].log_data[47].valid := 1, [127].log_data[48].min := 7.2114625, [127].log_data[48].max := 7.3296304, [127].log_data[48].total := 26066.104, [127].log_data[48].time := 3600.0, [127].log_data[48].minminute := 59, [127].log_data[48].maxminute := 27, [127].log_data[48].valid := 1, [127].log_data[49].min := 9.253142, [127].log_data[49].max := 9.377787, [127].log_data[49].total := 33467.85, [127].log_data[49].time := 3600.0, [127].log_data[49].minminute := 39, [127].log_data[49].maxminute := 54, [127].log_data[49].valid := 1, [127].log_data[50].min := 1.6079597, [127].log_data[50].max := 1.612553, [127].log_data[50].total := 5798.482, [127].log_data[50].time := 3600.0, [127].log_data[50].maxminute := 42, [127].log_data[50].valid := 1, [127].log_data[51].time := 3600.0, [127].log_data[51].valid := 1, [127].log_data[52].min := -1.6200027, [127].log_data[52].max := -1.4400024, [127].log_data[52].total := -5485.3315,
        [127].log_data[52].time := 3600.0, [127].log_data[52].minminute := 55, [127].log_data[52].valid := 1, [127].log_data[53].min := -1.5200043, [127].log_data[53].max := -1.340004, [127].log_data[53].total := -5173.416, [127].log_data[53].time := 3600.0, [127].log_data[53].minminute := 52, [127].log_data[53].maxminute := 1, [127].log_data[53].valid := 1, [127].log_data[54].time := 3600.0, [127].log_data[54].valid := 1, [127].log_data[55].time := 3600.0, [127].log_data[55].valid := 1, [127].log_data[56].min := 0.1592249, [127].log_data[56].max := 0.159696, [127].log_data[56].total := 573.9437, [127].log_data[56].time := 3600.0, [127].log_data[56].minminute := 54, [127].log_data[56].maxminute := 4, [127].log_data[56].valid := 1, [127].log_data[57].min := 0.20083867, [127].log_data[57].max := 0.20130977, [127].log_data[57].total := 723.7355, [127].log_data[57].time := 3600.0, [127].log_data[57].minminute := 1, [127].log_data[57].maxminute := 29, [127].log_data[57].valid := 1, [127].log_data[58].time := 3600.0, [127].log_data[58].valid := 1, [127].log_data[59].time := 3600.0, [127].log_data[59].valid := 1, [127].log_data[60].valid := 1, [127].log_data[61].valid := 1, [127].log_data[62].valid := 1, [127].log_data[63].valid := 1, [127].log_data[64].valid := 1, [127].log_data[65].valid := 1, [127].log_data[66].valid := 1, [127].log_data[67].valid := 1, [127].log_data[68].valid := 1, [127].log_data[69].valid := 1, [127].log_data[70].valid := 1, [127].log_data[71].valid := 1, [127].log_data[72].valid := 1, [127].log_data[73].valid := 1, [127].log_data[74].valid := 1, [127].log_data[75].valid := 1, [127].log_data[76].valid := 1, [127].log_data[77].valid := 1, [127].log_data[78].valid := 1, [127].log_data[79].valid := 1, [127].log_data[80].valid := 1, [127].log_data[81].valid := 1, [127].log_data[82].valid := 1, [127].log_data[83].valid := 1, [127].log_data[84].valid := 1, [127].log_data[85].valid := 1, [127].log_data[86].valid := 1, [127].log_data[87].valid := 1,
        [127].log_data[88].valid := 1, [127].log_data[89].valid := 1, [127].log_data[90].valid := 1, [127].log_data[91].valid := 1, [127].log_data[92].valid := 1, [127].log_data[93].valid := 1, [127].log_data[94].valid := 1, [127].log_data[95].valid := 1, [127].log_data[96].valid := 1, [127].log_data[97].valid := 1, [127].log_data[98].valid := 1, [127].log_data[99].valid := 1, [127].log_data[100].valid := 1, [127].log_data[101].valid := 1, [127].log_data[102].valid := 1, [127].log_data[103].valid := 1, [127].log_data[104].valid := 1, [127].log_data[105].valid := 1, [127].log_data[106].valid := 1, [127].log_data[107].valid := 1, [127].log_data[108].valid := 1, [127].log_data[109].valid := 1, [127].log_data[110].valid := 1, [127].log_data[111].valid := 1, [127].log_data[112].valid := 1, [127].log_data[113].valid := 1, [127].log_data[114].valid := 1, [127].log_data[115].valid := 1, [127].log_data[116].valid := 1, [127].log_data[117].valid := 1, [127].log_data[118].valid := 1, [127].log_data[119].valid := 1, [127].log_data[120].valid := 1, [127].log_data[121].valid := 1, [127].log_data[122].valid := 1, [127].log_data[123].valid := 1, [127].log_data[124].valid := 1, [127].time.Year := 2023, [127].time.Month := 1, [127].time.Day := 18, [127].time.Hour := 10, [127].time.Minute := 59, [127].time.Second := 59, [128].log_data[0].min := 1.0, [128].log_data[0].max := 1.0, [128].log_data[0].total := 3600.0, [128].log_data[0].time := 3600.0, [128].log_data[0].valid := 1, [128].log_data[1].max := 1.0, [128].log_data[1].total := 566.5, [128].log_data[1].time := 3600.0, [128].log_data[1].maxminute := 3, [128].log_data[1].valid := 1, [128].log_data[2].max := 1.0, [128].log_data[2].total := 563.0, [128].log_data[2].time := 3600.0, [128].log_data[2].maxminute := 3, [128].log_data[2].valid := 1, [128].log_data[3].time := 3600.0, [128].log_data[3].valid := 1,
        [128].log_data[4].time := 3600.0, [128].log_data[4].valid := 1, [128].log_data[5].max := 1.0, [128].log_data[5].total := 277.5, [128].log_data[5].time := 3600.0, [128].log_data[5].maxminute := 4, [128].log_data[5].valid := 1, [128].log_data[6].time := 3600.0, [128].log_data[6].valid := 1, [128].log_data[7].time := 3600.0, [128].log_data[7].valid := 1, [128].log_data[8].time := 3600.0, [128].log_data[8].valid := 1, [128].log_data[9].time := 3600.0, [128].log_data[9].valid := 1, [128].log_data[10].min := 1.0, [128].log_data[10].max := 1.0, [128].log_data[10].total := 3600.0, [128].log_data[10].time := 3600.0, [128].log_data[10].valid := 1, [128].log_data[11].time := 3600.0, [128].log_data[11].valid := 1, [128].log_data[12].min := 1.0, [128].log_data[12].max := 1.0, [128].log_data[12].total := 3600.0, [128].log_data[12].time := 3600.0, [128].log_data[12].valid := 1, [128].log_data[13].min := 1.0, [128].log_data[13].max := 1.0, [128].log_data[13].total := 3600.0, [128].log_data[13].time := 3600.0, [128].log_data[13].valid := 1, [128].log_data[14].time := 3600.0, [128].log_data[14].valid := 1, [128].log_data[15].time := 3600.0, [128].log_data[15].valid := 1, [128].log_data[16].time := 3600.0, [128].log_data[16].valid := 1, [128].log_data[17].min := 1.0, [128].log_data[17].max := 1.0, [128].log_data[17].total := 3600.0, [128].log_data[17].time := 3600.0, [128].log_data[17].valid := 1, [128].log_data[18].time := 3600.0, [128].log_data[18].valid := 1, [128].log_data[19].time := 3600.0, [128].log_data[19].valid := 1, [128].log_data[20].time := 3600.0, [128].log_data[20].valid := 1, [128].log_data[21].min := 1.0, [128].log_data[21].max := 1.0, [128].log_data[21].total := 3600.0, [128].log_data[21].time := 3600.0, [128].log_data[21].valid := 1, [128].log_data[22].time := 3600.0, [128].log_data[22].valid := 1, [128].log_data[23].time := 3600.0, [128].log_data[23].valid := 1, [128].log_data[24].time := 3600.0, [128].log_data[24].valid := 1,
        [128].log_data[25].time := 3600.0, [128].log_data[25].valid := 1, [128].log_data[26].time := 3600.0, [128].log_data[26].valid := 1, [128].log_data[27].time := 3600.0, [128].log_data[27].valid := 1, [128].log_data[28].time := 3600.0, [128].log_data[28].valid := 1, [128].log_data[29].min := 1.0, [128].log_data[29].max := 1.0, [128].log_data[29].total := 3600.0, [128].log_data[29].time := 3600.0, [128].log_data[29].valid := 1, [128].log_data[30].min := 1.0, [128].log_data[30].max := 1.0, [128].log_data[30].total := 3600.0, [128].log_data[30].time := 3600.0, [128].log_data[30].valid := 1, [128].log_data[31].time := 3600.0, [128].log_data[31].valid := 1, [128].log_data[32].time := 3600.0, [128].log_data[32].valid := 1, [128].log_data[33].time := 3600.0, [128].log_data[33].valid := 1, [128].log_data[34].time := 3600.0, [128].log_data[34].valid := 1, [128].log_data[35].time := 3600.0, [128].log_data[35].valid := 1, [128].log_data[36].time := 3600.0, [128].log_data[36].valid := 1, [128].log_data[37].max := 7.3172836, [128].log_data[37].total := 3597.804, [128].log_data[37].time := 3600.0, [128].log_data[37].maxminute := 4, [128].log_data[37].valid := 1, [128].log_data[38].time := 3600.0, [128].log_data[38].valid := 1, [128].log_data[39].min := 0.9982394, [128].log_data[39].max := 1.0221478, [128].log_data[39].total := 3621.872, [128].log_data[39].time := 3600.0, [128].log_data[39].minminute := 6, [128].log_data[39].maxminute := 9, [128].log_data[39].valid := 1, [128].log_data[40].min := 7.5997667, [128].log_data[40].max := 7.614607, [128].log_data[40].total := 27387.773, [128].log_data[40].time := 3600.0, [128].log_data[40].minminute := 38, [128].log_data[40].maxminute := 41, [128].log_data[40].valid := 1, [128].log_data[41].min := 0.022343751, [128].log_data[41].max := 0.022932617, [128].log_data[41].total := 81.7059, [128].log_data[41].time := 3600.0, [128].log_data[41].minminute := 34, [128].log_data[41].valid := 1, [128].log_data[42].min := 2.291407, [128].log_data[42].max := 2.2960005, [128].log_data[42].total := 8258.034,
        [128].log_data[42].time := 3600.0, [128].log_data[42].minminute := 16, [128].log_data[42].maxminute := 28, [128].log_data[42].valid := 1, [128].log_data[43].min := -0.26000214, [128].log_data[43].max := -0.23999786, [128].log_data[43].total := -935.6084, [128].log_data[43].time := 3600.0, [128].log_data[43].valid := 1, [128].log_data[44].min := -0.30000305, [128].log_data[44].max := -0.27999878, [128].log_data[44].total := -1035.9484, [128].log_data[44].time := 3600.0, [128].log_data[44].valid := 1, [128].log_data[45].time := 3600.0, [128].log_data[45].valid := 1, [128].log_data[46].time := 3600.0, [128].log_data[46].valid := 1, [128].log_data[47].time := 3600.0, [128].log_data[47].valid := 1, [128].log_data[48].min := 6.840198, [128].log_data[48].max := 7.278517, [128].log_data[48].total := 25347.986, [128].log_data[48].time := 3600.0, [128].log_data[48].minminute := 57, [128].log_data[48].maxminute := 5, [128].log_data[48].valid := 1, [128].log_data[49].min := 8.863308, [128].log_data[49].max := 9.307711, [128].log_data[49].total := 32804.45, [128].log_data[49].time := 3600.0, [128].log_data[49].minminute := 56, [128].log_data[49].maxminute := 59, [128].log_data[49].valid := 1, [128].log_data[50].min := 1.6103153, [128].log_data[50].max := 1.7555315, [128].log_data[50].total := 6237.0127, [128].log_data[50].time := 3600.0, [128].log_data[50].minminute := 1, [128].log_data[50].maxminute := 55, [128].log_data[50].valid := 1, [128].log_data[51].time := 3600.0, [128].log_data[51].valid := 1, [128].log_data[52].min := -1.6600037, [128].log_data[52].max := -1.4599991, [128].log_data[52].total := -5582.1646, [128].log_data[52].time := 3600.0, [128].log_data[52].minminute := 18, [128].log_data[52].maxminute := 36, [128].log_data[52].valid := 1, [128].log_data[53].min := -1.5400009, [128].log_data[53].max := -1.340004, [128].log_data[53].total := -5209.154, [128].log_data[53].time := 3600.0, [128].log_data[53].minminute := 16, [128].log_data[53].maxminute := 24, [128].log_data[53].valid := 1, [128].log_data[54].time := 3600.0, [128].log_data[54].valid := 1, [128].log_data[55].time := 3600.0,
        [128].log_data[55].valid := 1, [128].log_data[56].min := 0.15914638, [128].log_data[56].max := 0.15957822, [128].log_data[56].total := 573.55023, [128].log_data[56].time := 3600.0, [128].log_data[56].minminute := 12, [128].log_data[56].maxminute := 10, [128].log_data[56].valid := 1, [128].log_data[57].min := 0.20095645, [128].log_data[57].max := 0.20134902, [128].log_data[57].total := 723.97955, [128].log_data[57].time := 3600.0, [128].log_data[57].minminute := 10, [128].log_data[57].valid := 1, [128].log_data[58].time := 3600.0, [128].log_data[58].valid := 1, [128].log_data[59].time := 3600.0, [128].log_data[59].valid := 1, [128].log_data[60].valid := 1, [128].log_data[61].valid := 1, [128].log_data[62].valid := 1, [128].log_data[63].valid := 1, [128].log_data[64].valid := 1, [128].log_data[65].valid := 1, [128].log_data[66].valid := 1, [128].log_data[67].valid := 1, [128].log_data[68].valid := 1, [128].log_data[69].valid := 1, [128].log_data[70].valid := 1, [128].log_data[71].valid := 1, [128].log_data[72].valid := 1, [128].log_data[73].valid := 1, [128].log_data[74].valid := 1, [128].log_data[75].valid := 1, [128].log_data[76].valid := 1, [128].log_data[77].valid := 1, [128].log_data[78].valid := 1, [128].log_data[79].valid := 1, [128].log_data[80].valid := 1, [128].log_data[81].valid := 1, [128].log_data[82].valid := 1, [128].log_data[83].valid := 1, [128].log_data[84].valid := 1, [128].log_data[85].valid := 1, [128].log_data[86].valid := 1, [128].log_data[87].valid := 1, [128].log_data[88].valid := 1, [128].log_data[89].valid := 1, [128].log_data[90].valid := 1, [128].log_data[91].valid := 1, [128].log_data[92].valid := 1, [128].log_data[93].valid := 1, [128].log_data[94].valid := 1, [128].log_data[95].valid := 1, [128].log_data[96].valid := 1, [128].log_data[97].valid := 1, [128].log_data[98].valid := 1, [128].log_data[99].valid := 1, [128].log_data[100].valid := 1, [128].log_data[101].valid := 1,
        [128].log_data[102].valid := 1, [128].log_data[103].valid := 1, [128].log_data[104].valid := 1, [128].log_data[105].valid := 1, [128].log_data[106].valid := 1, [128].log_data[107].valid := 1, [128].log_data[108].valid := 1, [128].log_data[109].valid := 1, [128].log_data[110].valid := 1, [128].log_data[111].valid := 1, [128].log_data[112].valid := 1, [128].log_data[113].valid := 1, [128].log_data[114].valid := 1, [128].log_data[115].valid := 1, [128].log_data[116].valid := 1, [128].log_data[117].valid := 1, [128].log_data[118].valid := 1, [128].log_data[119].valid := 1, [128].log_data[120].valid := 1, [128].log_data[121].valid := 1, [128].log_data[122].valid := 1, [128].log_data[123].valid := 1, [128].log_data[124].valid := 1, [128].time.Year := 2023, [128].time.Month := 1, [128].time.Day := 18, [128].time.Hour := 11, [128].time.Minute := 59, [128].time.Second := 59, [129].log_data[0].min := 1.0, [129].log_data[0].max := 1.0, [129].log_data[0].total := 3600.0, [129].log_data[0].time := 3600.0, [129].log_data[0].valid := 1, [129].log_data[1].max := 1.0, [129].log_data[1].total := 535.5, [129].log_data[1].time := 3600.0, [129].log_data[1].maxminute := 42, [129].log_data[1].valid := 1, [129].log_data[2].max := 1.0, [129].log_data[2].total := 532.0, [129].log_data[2].time := 3600.0, [129].log_data[2].maxminute := 42, [129].log_data[2].valid := 1, [129].log_data[3].time := 3600.0, [129].log_data[3].valid := 1, [129].log_data[4].time := 3600.0, [129].log_data[4].valid := 1, [129].log_data[5].max := 1.0, [129].log_data[5].total := 251.5, [129].log_data[5].time := 3600.0, [129].log_data[5].maxminute := 44, [129].log_data[5].valid := 1, [129].log_data[6].time := 3600.0, [129].log_data[6].valid := 1, [129].log_data[7].time := 3600.0, [129].log_data[7].valid := 1, [129].log_data[8].time := 3600.0, [129].log_data[8].valid := 1, [129].log_data[9].time := 3600.0,
        [129].log_data[9].valid := 1, [129].log_data[10].min := 1.0, [129].log_data[10].max := 1.0, [129].log_data[10].total := 3600.0, [129].log_data[10].time := 3600.0, [129].log_data[10].valid := 1, [129].log_data[11].time := 3600.0, [129].log_data[11].valid := 1, [129].log_data[12].min := 1.0, [129].log_data[12].max := 1.0, [129].log_data[12].total := 3600.0, [129].log_data[12].time := 3600.0, [129].log_data[12].valid := 1, [129].log_data[13].min := 1.0, [129].log_data[13].max := 1.0, [129].log_data[13].total := 3600.0, [129].log_data[13].time := 3600.0, [129].log_data[13].valid := 1, [129].log_data[14].time := 3600.0, [129].log_data[14].valid := 1, [129].log_data[15].time := 3600.0, [129].log_data[15].valid := 1, [129].log_data[16].time := 3600.0, [129].log_data[16].valid := 1, [129].log_data[17].min := 1.0, [129].log_data[17].max := 1.0, [129].log_data[17].total := 3600.0, [129].log_data[17].time := 3600.0, [129].log_data[17].valid := 1, [129].log_data[18].time := 3600.0, [129].log_data[18].valid := 1, [129].log_data[19].time := 3600.0, [129].log_data[19].valid := 1, [129].log_data[20].time := 3600.0, [129].log_data[20].valid := 1, [129].log_data[21].min := 1.0, [129].log_data[21].max := 1.0, [129].log_data[21].total := 3600.0, [129].log_data[21].time := 3600.0, [129].log_data[21].valid := 1, [129].log_data[22].time := 3600.0, [129].log_data[22].valid := 1, [129].log_data[23].time := 3600.0, [129].log_data[23].valid := 1, [129].log_data[24].time := 3600.0, [129].log_data[24].valid := 1, [129].log_data[25].time := 3600.0, [129].log_data[25].valid := 1, [129].log_data[26].time := 3600.0, [129].log_data[26].valid := 1, [129].log_data[27].time := 3600.0, [129].log_data[27].valid := 1, [129].log_data[28].time := 3600.0, [129].log_data[28].valid := 1, [129].log_data[29].min := 1.0, [129].log_data[29].max := 1.0, [129].log_data[29].total := 3600.0, [129].log_data[29].time := 3600.0, [129].log_data[29].valid := 1, [129].log_data[30].min := 1.0,
        [129].log_data[30].max := 1.0, [129].log_data[30].total := 3600.0, [129].log_data[30].time := 3600.0, [129].log_data[30].valid := 1, [129].log_data[31].time := 3600.0, [129].log_data[31].valid := 1, [129].log_data[32].time := 3600.0, [129].log_data[32].valid := 1, [129].log_data[33].time := 3600.0, [129].log_data[33].valid := 1, [129].log_data[34].time := 3600.0, [129].log_data[34].valid := 1, [129].log_data[35].time := 3600.0, [129].log_data[35].valid := 1, [129].log_data[36].time := 3600.0, [129].log_data[36].valid := 1, [129].log_data[37].max := 7.5759954, [129].log_data[37].total := 3513.0034, [129].log_data[37].time := 3600.0, [129].log_data[37].maxminute := 45, [129].log_data[37].valid := 1, [129].log_data[38].time := 3600.0, [129].log_data[38].valid := 1, [129].log_data[39].min := 0.9961195, [129].log_data[39].max := 1.0225011, [129].log_data[39].total := 3619.3274, [129].log_data[39].time := 3600.0, [129].log_data[39].minminute := 51, [129].log_data[39].maxminute := 49, [129].log_data[39].valid := 1, [129].log_data[40].min := 7.5871253, [129].log_data[40].max := 7.621752, [129].log_data[40].total := 27385.379, [129].log_data[40].time := 3600.0, [129].log_data[40].minminute := 29, [129].log_data[40].maxminute := 36, [129].log_data[40].valid := 1, [129].log_data[41].min := 0.022343751, [129].log_data[41].max := 0.022932617, [129].log_data[41].total := 81.688965, [129].log_data[41].time := 3600.0, [129].log_data[41].minminute := 1, [129].log_data[41].valid := 1, [129].log_data[42].min := 2.2912893, [129].log_data[42].max := 2.2958827, [129].log_data[42].total := 8258.141, [129].log_data[42].time := 3600.0, [129].log_data[42].minminute := 53, [129].log_data[42].maxminute := 11, [129].log_data[42].valid := 1, [129].log_data[43].min := -0.26000214, [129].log_data[43].max := -0.23999786, [129].log_data[43].total := -935.3876, [129].log_data[43].time := 3600.0, [129].log_data[43].maxminute := 1, [129].log_data[43].valid := 1, [129].log_data[44].min := -0.30000305, [129].log_data[44].max := -0.27999878, [129].log_data[44].total := -1012.42163, [129].log_data[44].time := 3600.0,
        [129].log_data[44].valid := 1, [129].log_data[45].time := 3600.0, [129].log_data[45].valid := 1, [129].log_data[46].time := 3600.0, [129].log_data[46].valid := 1, [129].log_data[47].time := 3600.0, [129].log_data[47].valid := 1, [129].log_data[48].min := 6.847068, [129].log_data[48].max := 7.041907, [129].log_data[48].total := 24903.34, [129].log_data[48].time := 3600.0, [129].log_data[48].maxminute := 47, [129].log_data[48].valid := 1, [129].log_data[49].min := 6.5796537, [129].log_data[49].max := 9.505966, [129].log_data[49].total := 32593.848, [129].log_data[49].time := 3600.0, [129].log_data[49].minminute := 59, [129].log_data[49].maxminute := 40, [129].log_data[49].valid := 1, [129].log_data[50].min := 1.751174, [129].log_data[50].max := 1.8820219, [129].log_data[50].total := 6405.6685, [129].log_data[50].time := 3600.0, [129].log_data[50].minminute := 3, [129].log_data[50].maxminute := 58, [129].log_data[50].valid := 1, [129].log_data[51].time := 3600.0, [129].log_data[51].valid := 1, [129].log_data[52].min := -1.6200027, [129].log_data[52].max := -1.4599991, [129].log_data[52].total := -5554.051, [129].log_data[52].time := 3600.0, [129].log_data[52].minminute := 4, [129].log_data[52].maxminute := 52, [129].log_data[52].valid := 1, [129].log_data[53].min := -1.5400009, [129].log_data[53].max := -1.4000015, [129].log_data[53].total := -5239.5063, [129].log_data[53].time := 3600.0, [129].log_data[53].minminute := 6, [129].log_data[53].maxminute := 10, [129].log_data[53].valid := 1, [129].log_data[54].time := 3600.0, [129].log_data[54].valid := 1, [129].log_data[55].time := 3600.0, [129].log_data[55].valid := 1, [129].log_data[56].min := 0.15914638, [129].log_data[56].max := 0.15953897, [129].log_data[56].total := 573.4412, [129].log_data[56].time := 3600.0, [129].log_data[56].minminute := 10, [129].log_data[56].maxminute := 5, [129].log_data[56].valid := 1, [129].log_data[57].min := 0.2009957, [129].log_data[57].max := 0.20138828, [129].log_data[57].total := 724.1213, [129].log_data[57].time := 3600.0, [129].log_data[57].minminute := 20, [129].log_data[57].maxminute := 12,
        [129].log_data[57].valid := 1, [129].log_data[58].time := 3600.0, [129].log_data[58].valid := 1, [129].log_data[59].time := 3600.0, [129].log_data[59].valid := 1, [129].log_data[60].valid := 1, [129].log_data[61].valid := 1, [129].log_data[62].valid := 1, [129].log_data[63].valid := 1, [129].log_data[64].valid := 1, [129].log_data[65].valid := 1, [129].log_data[66].valid := 1, [129].log_data[67].valid := 1, [129].log_data[68].valid := 1, [129].log_data[69].valid := 1, [129].log_data[70].valid := 1, [129].log_data[71].valid := 1, [129].log_data[72].valid := 1, [129].log_data[73].valid := 1, [129].log_data[74].valid := 1, [129].log_data[75].valid := 1, [129].log_data[76].valid := 1, [129].log_data[77].valid := 1, [129].log_data[78].valid := 1, [129].log_data[79].valid := 1, [129].log_data[80].valid := 1, [129].log_data[81].valid := 1, [129].log_data[82].valid := 1, [129].log_data[83].valid := 1, [129].log_data[84].valid := 1, [129].log_data[85].valid := 1, [129].log_data[86].valid := 1, [129].log_data[87].valid := 1, [129].log_data[88].valid := 1, [129].log_data[89].valid := 1, [129].log_data[90].valid := 1, [129].log_data[91].valid := 1, [129].log_data[92].valid := 1, [129].log_data[93].valid := 1, [129].log_data[94].valid := 1, [129].log_data[95].valid := 1, [129].log_data[96].valid := 1, [129].log_data[97].valid := 1, [129].log_data[98].valid := 1, [129].log_data[99].valid := 1, [129].log_data[100].valid := 1, [129].log_data[101].valid := 1, [129].log_data[102].valid := 1, [129].log_data[103].valid := 1, [129].log_data[104].valid := 1, [129].log_data[105].valid := 1, [129].log_data[106].valid := 1, [129].log_data[107].valid := 1, [129].log_data[108].valid := 1, [129].log_data[109].valid := 1, [129].log_data[110].valid := 1, [129].log_data[111].valid := 1, [129].log_data[112].valid := 1, [129].log_data[113].valid := 1, [129].log_data[114].valid := 1,
        [129].log_data[115].valid := 1, [129].log_data[116].valid := 1, [129].log_data[117].valid := 1, [129].log_data[118].valid := 1, [129].log_data[119].valid := 1, [129].log_data[120].valid := 1, [129].log_data[121].valid := 1, [129].log_data[122].valid := 1, [129].log_data[123].valid := 1, [129].log_data[124].valid := 1, [129].time.Year := 2023, [129].time.Month := 1, [129].time.Day := 18, [129].time.Hour := 12, [129].time.Minute := 59, [129].time.Second := 59, [130].log_data[0].min := 1.0, [130].log_data[0].max := 1.0, [130].log_data[0].total := 3600.0, [130].log_data[0].time := 3600.0, [130].log_data[0].valid := 1, [130].log_data[1].time := 3600.0, [130].log_data[1].valid := 1, [130].log_data[2].time := 3600.0, [130].log_data[2].valid := 1, [130].log_data[3].time := 3600.0, [130].log_data[3].valid := 1, [130].log_data[4].time := 3600.0, [130].log_data[4].valid := 1, [130].log_data[5].time := 3600.0, [130].log_data[5].valid := 1, [130].log_data[6].time := 3600.0, [130].log_data[6].valid := 1, [130].log_data[7].time := 3600.0, [130].log_data[7].valid := 1, [130].log_data[8].time := 3600.0, [130].log_data[8].valid := 1, [130].log_data[9].time := 3600.0, [130].log_data[9].valid := 1, [130].log_data[10].min := 1.0, [130].log_data[10].max := 1.0, [130].log_data[10].total := 3600.0, [130].log_data[10].time := 3600.0, [130].log_data[10].valid := 1, [130].log_data[11].time := 3600.0, [130].log_data[11].valid := 1, [130].log_data[12].min := 1.0, [130].log_data[12].max := 1.0, [130].log_data[12].total := 3600.0, [130].log_data[12].time := 3600.0, [130].log_data[12].valid := 1, [130].log_data[13].min := 1.0, [130].log_data[13].max := 1.0, [130].log_data[13].total := 3600.0, [130].log_data[13].time := 3600.0, [130].log_data[13].valid := 1, [130].log_data[14].time := 3600.0, [130].log_data[14].valid := 1, [130].log_data[15].time := 3600.0, [130].log_data[15].valid := 1,
        [130].log_data[16].time := 3600.0, [130].log_data[16].valid := 1, [130].log_data[17].min := 1.0, [130].log_data[17].max := 1.0, [130].log_data[17].total := 3600.0, [130].log_data[17].time := 3600.0, [130].log_data[17].valid := 1, [130].log_data[18].time := 3600.0, [130].log_data[18].valid := 1, [130].log_data[19].time := 3600.0, [130].log_data[19].valid := 1, [130].log_data[20].time := 3600.0, [130].log_data[20].valid := 1, [130].log_data[21].min := 1.0, [130].log_data[21].max := 1.0, [130].log_data[21].total := 3600.0, [130].log_data[21].time := 3600.0, [130].log_data[21].valid := 1, [130].log_data[22].time := 3600.0, [130].log_data[22].valid := 1, [130].log_data[23].time := 3600.0, [130].log_data[23].valid := 1, [130].log_data[24].time := 3600.0, [130].log_data[24].valid := 1, [130].log_data[25].time := 3600.0, [130].log_data[25].valid := 1, [130].log_data[26].time := 3600.0, [130].log_data[26].valid := 1, [130].log_data[27].time := 3600.0, [130].log_data[27].valid := 1, [130].log_data[28].time := 3600.0, [130].log_data[28].valid := 1, [130].log_data[29].min := 1.0, [130].log_data[29].max := 1.0, [130].log_data[29].total := 3600.0, [130].log_data[29].time := 3600.0, [130].log_data[29].valid := 1, [130].log_data[30].min := 1.0, [130].log_data[30].max := 1.0, [130].log_data[30].total := 3600.0, [130].log_data[30].time := 3600.0, [130].log_data[30].valid := 1, [130].log_data[31].time := 3600.0, [130].log_data[31].valid := 1, [130].log_data[32].time := 3600.0, [130].log_data[32].valid := 1, [130].log_data[33].time := 3600.0, [130].log_data[33].valid := 1, [130].log_data[34].time := 3600.0, [130].log_data[34].valid := 1, [130].log_data[35].time := 3600.0, [130].log_data[35].valid := 1, [130].log_data[36].time := 3600.0, [130].log_data[36].valid := 1, [130].log_data[37].time := 3600.0, [130].log_data[37].valid := 1, [130].log_data[38].time := 3600.0, [130].log_data[38].valid := 1, [130].log_data[39].min := 0.9961195, [130].log_data[39].max := 1.0048349,
        [130].log_data[39].total := 3604.882, [130].log_data[39].time := 3600.0, [130].log_data[39].minminute := 41, [130].log_data[39].maxminute := 59, [130].log_data[39].valid := 1, [130].log_data[40].min := 7.6025147, [130].log_data[40].max := 7.6132326, [130].log_data[40].total := 27389.42, [130].log_data[40].time := 3600.0, [130].log_data[40].minminute := 30, [130].log_data[40].maxminute := 34, [130].log_data[40].valid := 1, [130].log_data[41].min := 0.022343751, [130].log_data[41].max := 0.022932617, [130].log_data[41].total := 81.51651, [130].log_data[41].time := 3600.0, [130].log_data[41].minminute := 4, [130].log_data[41].maxminute := 3, [130].log_data[41].valid := 1, [130].log_data[42].min := 2.2912893, [130].log_data[42].max := 2.2957647, [130].log_data[42].total := 8257.894, [130].log_data[42].time := 3600.0, [130].log_data[42].minminute := 27, [130].log_data[42].maxminute := 35, [130].log_data[42].valid := 1, [130].log_data[43].min := -0.26000214, [130].log_data[43].max := -0.23999786, [130].log_data[43].total := -935.6831, [130].log_data[43].time := 3600.0, [130].log_data[43].valid := 1, [130].log_data[44].min := -0.30000305, [130].log_data[44].max := -0.27999878, [130].log_data[44].total := -1010.936, [130].log_data[44].time := 3600.0, [130].log_data[44].minminute := 1, [130].log_data[44].valid := 1, [130].log_data[45].time := 3600.0, [130].log_data[45].valid := 1, [130].log_data[46].time := 3600.0, [130].log_data[46].valid := 1, [130].log_data[47].time := 3600.0, [130].log_data[47].valid := 1, [130].log_data[48].min := 6.717084, [130].log_data[48].max := 6.9176936, [130].log_data[48].total := 24414.193, [130].log_data[48].time := 3600.0, [130].log_data[48].minminute := 34, [130].log_data[48].valid := 1, [130].log_data[49].min := 5.2158213, [130].log_data[49].max := 8.477595, [130].log_data[49].total := 22798.637, [130].log_data[49].time := 3600.0, [130].log_data[49].minminute := 25, [130].log_data[49].maxminute := 59, [130].log_data[49].valid := 1, [130].log_data[50].min := 1.8753086, [130].log_data[50].max := 1.8861439, [130].log_data[50].total := 6777.145, [130].log_data[50].time := 3600.0,
        [130].log_data[50].minminute := 1, [130].log_data[50].maxminute := 38, [130].log_data[50].valid := 1, [130].log_data[51].time := 3600.0, [130].log_data[51].valid := 1, [130].log_data[52].min := -1.6200027, [130].log_data[52].max := -1.4599991, [130].log_data[52].total := -5600.6333, [130].log_data[52].time := 3600.0, [130].log_data[52].minminute := 6, [130].log_data[52].maxminute := 1, [130].log_data[52].valid := 1, [130].log_data[53].min := -1.5400009, [130].log_data[53].max := -1.4000015, [130].log_data[53].total := -5265.693, [130].log_data[53].time := 3600.0, [130].log_data[53].minminute := 1, [130].log_data[53].maxminute := 34, [130].log_data[53].valid := 1, [130].log_data[54].time := 3600.0, [130].log_data[54].valid := 1, [130].log_data[55].time := 3600.0, [130].log_data[55].valid := 1, [130].log_data[56].min := 0.15906787, [130].log_data[56].max := 0.15942119, [130].log_data[56].total := 573.1499, [130].log_data[56].time := 3600.0, [130].log_data[56].minminute := 6, [130].log_data[56].valid := 1, [130].log_data[57].min := 0.2009957, [130].log_data[57].max := 0.20138828, [130].log_data[57].total := 724.13794, [130].log_data[57].time := 3600.0, [130].log_data[57].minminute := 4, [130].log_data[57].maxminute := 55, [130].log_data[57].valid := 1, [130].log_data[58].time := 3600.0, [130].log_data[58].valid := 1, [130].log_data[59].time := 3600.0, [130].log_data[59].valid := 1, [130].log_data[60].valid := 1, [130].log_data[61].valid := 1, [130].log_data[62].valid := 1, [130].log_data[63].valid := 1, [130].log_data[64].valid := 1, [130].log_data[65].valid := 1, [130].log_data[66].valid := 1, [130].log_data[67].valid := 1, [130].log_data[68].valid := 1, [130].log_data[69].valid := 1, [130].log_data[70].valid := 1, [130].log_data[71].valid := 1, [130].log_data[72].valid := 1, [130].log_data[73].valid := 1, [130].log_data[74].valid := 1, [130].log_data[75].valid := 1, [130].log_data[76].valid := 1, [130].log_data[77].valid := 1, [130].log_data[78].valid := 1, [130].log_data[79].valid := 1,
        [130].log_data[80].valid := 1, [130].log_data[81].valid := 1, [130].log_data[82].valid := 1, [130].log_data[83].valid := 1, [130].log_data[84].valid := 1, [130].log_data[85].valid := 1, [130].log_data[86].valid := 1, [130].log_data[87].valid := 1, [130].log_data[88].valid := 1, [130].log_data[89].valid := 1, [130].log_data[90].valid := 1, [130].log_data[91].valid := 1, [130].log_data[92].valid := 1, [130].log_data[93].valid := 1, [130].log_data[94].valid := 1, [130].log_data[95].valid := 1, [130].log_data[96].valid := 1, [130].log_data[97].valid := 1, [130].log_data[98].valid := 1, [130].log_data[99].valid := 1, [130].log_data[100].valid := 1, [130].log_data[101].valid := 1, [130].log_data[102].valid := 1, [130].log_data[103].valid := 1, [130].log_data[104].valid := 1, [130].log_data[105].valid := 1, [130].log_data[106].valid := 1, [130].log_data[107].valid := 1, [130].log_data[108].valid := 1, [130].log_data[109].valid := 1, [130].log_data[110].valid := 1, [130].log_data[111].valid := 1, [130].log_data[112].valid := 1, [130].log_data[113].valid := 1, [130].log_data[114].valid := 1, [130].log_data[115].valid := 1, [130].log_data[116].valid := 1, [130].log_data[117].valid := 1, [130].log_data[118].valid := 1, [130].log_data[119].valid := 1, [130].log_data[120].valid := 1, [130].log_data[121].valid := 1, [130].log_data[122].valid := 1, [130].log_data[123].valid := 1, [130].log_data[124].valid := 1, [130].time.Year := 2023, [130].time.Month := 1, [130].time.Day := 18, [130].time.Hour := 13, [130].time.Minute := 59, [130].time.Second := 59, [131].log_data[0].min := 1.0, [131].log_data[0].max := 1.0, [131].log_data[0].total := 3600.0, [131].log_data[0].time := 3600.0, [131].log_data[0].valid := 1, [131].log_data[1].max := 1.0, [131].log_data[1].total := 558.5, [131].log_data[1].time := 3600.0, [131].log_data[1].maxminute := 35,
        [131].log_data[1].valid := 1, [131].log_data[2].max := 1.0, [131].log_data[2].total := 555.0, [131].log_data[2].time := 3600.0, [131].log_data[2].maxminute := 35, [131].log_data[2].valid := 1, [131].log_data[3].time := 3600.0, [131].log_data[3].valid := 1, [131].log_data[4].time := 3600.0, [131].log_data[4].valid := 1, [131].log_data[5].max := 1.0, [131].log_data[5].total := 240.0, [131].log_data[5].time := 3600.0, [131].log_data[5].maxminute := 38, [131].log_data[5].valid := 1, [131].log_data[6].time := 3600.0, [131].log_data[6].valid := 1, [131].log_data[7].time := 3600.0, [131].log_data[7].valid := 1, [131].log_data[8].time := 3600.0, [131].log_data[8].valid := 1, [131].log_data[9].time := 3600.0, [131].log_data[9].valid := 1, [131].log_data[10].min := 1.0, [131].log_data[10].max := 1.0, [131].log_data[10].total := 3600.0, [131].log_data[10].time := 3600.0, [131].log_data[10].valid := 1, [131].log_data[11].time := 3600.0, [131].log_data[11].valid := 1, [131].log_data[12].min := 1.0, [131].log_data[12].max := 1.0, [131].log_data[12].total := 3600.0, [131].log_data[12].time := 3600.0, [131].log_data[12].valid := 1, [131].log_data[13].min := 1.0, [131].log_data[13].max := 1.0, [131].log_data[13].total := 3600.0, [131].log_data[13].time := 3600.0, [131].log_data[13].valid := 1, [131].log_data[14].time := 3600.0, [131].log_data[14].valid := 1, [131].log_data[15].time := 3600.0, [131].log_data[15].valid := 1, [131].log_data[16].time := 3600.0, [131].log_data[16].valid := 1, [131].log_data[17].min := 1.0, [131].log_data[17].max := 1.0, [131].log_data[17].total := 3600.0, [131].log_data[17].time := 3600.0, [131].log_data[17].valid := 1, [131].log_data[18].time := 3600.0, [131].log_data[18].valid := 1, [131].log_data[19].time := 3600.0, [131].log_data[19].valid := 1, [131].log_data[20].time := 3600.0, [131].log_data[20].valid := 1, [131].log_data[21].min := 1.0, [131].log_data[21].max := 1.0, [131].log_data[21].total := 3600.0,
        [131].log_data[21].time := 3600.0, [131].log_data[21].valid := 1, [131].log_data[22].time := 3600.0, [131].log_data[22].valid := 1, [131].log_data[23].time := 3600.0, [131].log_data[23].valid := 1, [131].log_data[24].time := 3600.0, [131].log_data[24].valid := 1, [131].log_data[25].time := 3600.0, [131].log_data[25].valid := 1, [131].log_data[26].time := 3600.0, [131].log_data[26].valid := 1, [131].log_data[27].time := 3600.0, [131].log_data[27].valid := 1, [131].log_data[28].time := 3600.0, [131].log_data[28].valid := 1, [131].log_data[29].min := 1.0, [131].log_data[29].max := 1.0, [131].log_data[29].total := 3600.0, [131].log_data[29].time := 3600.0, [131].log_data[29].valid := 1, [131].log_data[30].min := 1.0, [131].log_data[30].max := 1.0, [131].log_data[30].total := 3600.0, [131].log_data[30].time := 3600.0, [131].log_data[30].valid := 1, [131].log_data[31].time := 3600.0, [131].log_data[31].valid := 1, [131].log_data[32].time := 3600.0, [131].log_data[32].valid := 1, [131].log_data[33].time := 3600.0, [131].log_data[33].valid := 1, [131].log_data[34].time := 3600.0, [131].log_data[34].valid := 1, [131].log_data[35].time := 3600.0, [131].log_data[35].valid := 1, [131].log_data[36].time := 3600.0, [131].log_data[36].valid := 1, [131].log_data[37].max := 7.1999016, [131].log_data[37].total := 3481.4167, [131].log_data[37].time := 3600.0, [131].log_data[37].maxminute := 36, [131].log_data[37].valid := 1, [131].log_data[38].time := 3600.0, [131].log_data[38].valid := 1, [131].log_data[39].min := 0.99635506, [131].log_data[39].max := 1.02097, [131].log_data[39].total := 3608.989, [131].log_data[39].time := 3600.0, [131].log_data[39].minminute := 5, [131].log_data[39].maxminute := 43, [131].log_data[39].valid := 1, [131].log_data[40].min := 7.602789, [131].log_data[40].max := 7.614332, [131].log_data[40].total := 27391.629, [131].log_data[40].time := 3600.0, [131].log_data[40].minminute := 29, [131].log_data[40].maxminute := 50, [131].log_data[40].valid := 1, [131].log_data[41].min := 0.022343751,
        [131].log_data[41].max := 0.022932617, [131].log_data[41].total := 81.67933, [131].log_data[41].time := 3600.0, [131].log_data[41].minminute := 4, [131].log_data[41].maxminute := 1, [131].log_data[41].valid := 1, [131].log_data[42].min := 2.2911716, [131].log_data[42].max := 2.2958827, [131].log_data[42].total := 8257.979, [131].log_data[42].time := 3600.0, [131].log_data[42].minminute := 23, [131].log_data[42].maxminute := 27, [131].log_data[42].valid := 1, [131].log_data[43].min := -0.26000214, [131].log_data[43].max := -0.23999786, [131].log_data[43].total := -935.0896, [131].log_data[43].time := 3600.0, [131].log_data[43].maxminute := 14, [131].log_data[43].valid := 1, [131].log_data[44].min := -0.30000305, [131].log_data[44].max := -0.27999878, [131].log_data[44].total := -1011.5348, [131].log_data[44].time := 3600.0, [131].log_data[44].valid := 1, [131].log_data[45].time := 3600.0, [131].log_data[45].valid := 1, [131].log_data[46].time := 3600.0, [131].log_data[46].valid := 1, [131].log_data[47].time := 3600.0, [131].log_data[47].valid := 1, [131].log_data[48].min := 6.7901826, [131].log_data[48].max := 7.0089297, [131].log_data[48].total := 24679.357, [131].log_data[48].time := 3600.0, [131].log_data[48].maxminute := 45, [131].log_data[48].valid := 1, [131].log_data[49].min := 6.4177136, [131].log_data[49].max := 9.364439, [131].log_data[49].total := 30918.916, [131].log_data[49].time := 3600.0, [131].log_data[49].minminute := 59, [131].log_data[49].maxminute := 38, [131].log_data[49].valid := 1, [131].log_data[50].min := 1.878253, [131].log_data[50].max := 2.0076876, [131].log_data[50].total := 6914.968, [131].log_data[50].time := 3600.0, [131].log_data[50].minminute := 24, [131].log_data[50].maxminute := 56, [131].log_data[50].valid := 1, [131].log_data[51].time := 3600.0, [131].log_data[51].valid := 1, [131].log_data[52].min := -1.6399994, [131].log_data[52].max := -1.4599991, [131].log_data[52].total := -5626.001, [131].log_data[52].time := 3600.0, [131].log_data[52].minminute := 5, [131].log_data[52].maxminute := 44, [131].log_data[52].valid := 1, [131].log_data[53].min := -1.5600052,
        [131].log_data[53].max := -1.4000015, [131].log_data[53].total := -5296.995, [131].log_data[53].time := 3600.0, [131].log_data[53].minminute := 50, [131].log_data[53].maxminute := 5, [131].log_data[53].valid := 1, [131].log_data[54].time := 3600.0, [131].log_data[54].valid := 1, [131].log_data[55].time := 3600.0, [131].log_data[55].valid := 1, [131].log_data[56].min := 0.15902862, [131].log_data[56].max := 0.15942119, [131].log_data[56].total := 573.11804, [131].log_data[56].time := 3600.0, [131].log_data[56].minminute := 55, [131].log_data[56].maxminute := 1, [131].log_data[56].valid := 1, [131].log_data[57].min := 0.20103496, [131].log_data[57].max := 0.20142753, [131].log_data[57].total := 724.20074, [131].log_data[57].time := 3600.0, [131].log_data[57].minminute := 5, [131].log_data[57].maxminute := 28, [131].log_data[57].valid := 1, [131].log_data[58].time := 3600.0, [131].log_data[58].valid := 1, [131].log_data[59].time := 3600.0, [131].log_data[59].valid := 1, [131].log_data[60].valid := 1, [131].log_data[61].valid := 1, [131].log_data[62].valid := 1, [131].log_data[63].valid := 1, [131].log_data[64].valid := 1, [131].log_data[65].valid := 1, [131].log_data[66].valid := 1, [131].log_data[67].valid := 1, [131].log_data[68].valid := 1, [131].log_data[69].valid := 1, [131].log_data[70].valid := 1, [131].log_data[71].valid := 1, [131].log_data[72].valid := 1, [131].log_data[73].valid := 1, [131].log_data[74].valid := 1, [131].log_data[75].valid := 1, [131].log_data[76].valid := 1, [131].log_data[77].valid := 1, [131].log_data[78].valid := 1, [131].log_data[79].valid := 1, [131].log_data[80].valid := 1, [131].log_data[81].valid := 1, [131].log_data[82].valid := 1, [131].log_data[83].valid := 1, [131].log_data[84].valid := 1, [131].log_data[85].valid := 1, [131].log_data[86].valid := 1, [131].log_data[87].valid := 1, [131].log_data[88].valid := 1, [131].log_data[89].valid := 1, [131].log_data[90].valid := 1, [131].log_data[91].valid := 1,
        [131].log_data[92].valid := 1, [131].log_data[93].valid := 1, [131].log_data[94].valid := 1, [131].log_data[95].valid := 1, [131].log_data[96].valid := 1, [131].log_data[97].valid := 1, [131].log_data[98].valid := 1, [131].log_data[99].valid := 1, [131].log_data[100].valid := 1, [131].log_data[101].valid := 1, [131].log_data[102].valid := 1, [131].log_data[103].valid := 1, [131].log_data[104].valid := 1, [131].log_data[105].valid := 1, [131].log_data[106].valid := 1, [131].log_data[107].valid := 1, [131].log_data[108].valid := 1, [131].log_data[109].valid := 1, [131].log_data[110].valid := 1, [131].log_data[111].valid := 1, [131].log_data[112].valid := 1, [131].log_data[113].valid := 1, [131].log_data[114].valid := 1, [131].log_data[115].valid := 1, [131].log_data[116].valid := 1, [131].log_data[117].valid := 1, [131].log_data[118].valid := 1, [131].log_data[119].valid := 1, [131].log_data[120].valid := 1, [131].log_data[121].valid := 1, [131].log_data[122].valid := 1, [131].log_data[123].valid := 1, [131].log_data[124].valid := 1, [131].time.Year := 2023, [131].time.Month := 1, [131].time.Day := 18, [131].time.Hour := 14, [131].time.Minute := 59, [131].time.Second := 59, [132].log_data[0].min := 1.0, [132].log_data[0].max := 1.0, [132].log_data[0].total := 3600.0, [132].log_data[0].time := 3600.0, [132].log_data[0].valid := 1, [132].log_data[1].time := 3600.0, [132].log_data[1].valid := 1, [132].log_data[2].time := 3600.0, [132].log_data[2].valid := 1, [132].log_data[3].time := 3600.0, [132].log_data[3].valid := 1, [132].log_data[4].time := 3600.0, [132].log_data[4].valid := 1, [132].log_data[5].time := 3600.0, [132].log_data[5].valid := 1, [132].log_data[6].time := 3600.0, [132].log_data[6].valid := 1, [132].log_data[7].time := 3600.0, [132].log_data[7].valid := 1, [132].log_data[8].time := 3600.0, [132].log_data[8].valid := 1,
        [132].log_data[9].time := 3600.0, [132].log_data[9].valid := 1, [132].log_data[10].min := 1.0, [132].log_data[10].max := 1.0, [132].log_data[10].total := 3600.0, [132].log_data[10].time := 3600.0, [132].log_data[10].valid := 1, [132].log_data[11].time := 3600.0, [132].log_data[11].valid := 1, [132].log_data[12].min := 1.0, [132].log_data[12].max := 1.0, [132].log_data[12].total := 3600.0, [132].log_data[12].time := 3600.0, [132].log_data[12].valid := 1, [132].log_data[13].min := 1.0, [132].log_data[13].max := 1.0, [132].log_data[13].total := 3600.0, [132].log_data[13].time := 3600.0, [132].log_data[13].valid := 1, [132].log_data[14].time := 3600.0, [132].log_data[14].valid := 1, [132].log_data[15].time := 3600.0, [132].log_data[15].valid := 1, [132].log_data[16].time := 3600.0, [132].log_data[16].valid := 1, [132].log_data[17].min := 1.0, [132].log_data[17].max := 1.0, [132].log_data[17].total := 3600.0, [132].log_data[17].time := 3600.0, [132].log_data[17].valid := 1, [132].log_data[18].time := 3600.0, [132].log_data[18].valid := 1, [132].log_data[19].time := 3600.0, [132].log_data[19].valid := 1, [132].log_data[20].time := 3600.0, [132].log_data[20].valid := 1, [132].log_data[21].min := 1.0, [132].log_data[21].max := 1.0, [132].log_data[21].total := 3600.0, [132].log_data[21].time := 3600.0, [132].log_data[21].valid := 1, [132].log_data[22].time := 3600.0, [132].log_data[22].valid := 1, [132].log_data[23].time := 3600.0, [132].log_data[23].valid := 1, [132].log_data[24].time := 3600.0, [132].log_data[24].valid := 1, [132].log_data[25].time := 3600.0, [132].log_data[25].valid := 1, [132].log_data[26].time := 3600.0, [132].log_data[26].valid := 1, [132].log_data[27].time := 3600.0, [132].log_data[27].valid := 1, [132].log_data[28].time := 3600.0, [132].log_data[28].valid := 1, [132].log_data[29].min := 1.0, [132].log_data[29].max := 1.0, [132].log_data[29].total := 3600.0, [132].log_data[29].time := 3600.0, [132].log_data[29].valid := 1,
        [132].log_data[30].min := 1.0, [132].log_data[30].max := 1.0, [132].log_data[30].total := 3600.0, [132].log_data[30].time := 3600.0, [132].log_data[30].valid := 1, [132].log_data[31].time := 3600.0, [132].log_data[31].valid := 1, [132].log_data[32].time := 3600.0, [132].log_data[32].valid := 1, [132].log_data[33].time := 3600.0, [132].log_data[33].valid := 1, [132].log_data[34].time := 3600.0, [132].log_data[34].valid := 1, [132].log_data[35].time := 3600.0, [132].log_data[35].valid := 1, [132].log_data[36].time := 3600.0, [132].log_data[36].valid := 1, [132].log_data[37].time := 3600.0, [132].log_data[37].valid := 1, [132].log_data[38].time := 3600.0, [132].log_data[38].valid := 1, [132].log_data[39].min := 0.995884, [132].log_data[39].max := 1.0040104, [132].log_data[39].total := 3600.835, [132].log_data[39].time := 3600.0, [132].log_data[39].minminute := 43, [132].log_data[39].maxminute := 5, [132].log_data[39].valid := 1, [132].log_data[40].min := 7.581355, [132].log_data[40].max := 7.617355, [132].log_data[40].total := 27386.47, [132].log_data[40].time := 3600.0, [132].log_data[40].minminute := 55, [132].log_data[40].maxminute := 22, [132].log_data[40].valid := 1, [132].log_data[41].min := 0.022343751, [132].log_data[41].max := 0.022932617, [132].log_data[41].total := 81.58355, [132].log_data[41].time := 3600.0, [132].log_data[41].minminute := 8, [132].log_data[41].valid := 1, [132].log_data[42].min := 2.2912893, [132].log_data[42].max := 2.2958827, [132].log_data[42].total := 8257.946, [132].log_data[42].time := 3600.0, [132].log_data[42].minminute := 53, [132].log_data[42].maxminute := 15, [132].log_data[42].valid := 1, [132].log_data[43].min := -0.26000214, [132].log_data[43].max := -0.23999786, [132].log_data[43].total := -934.7287, [132].log_data[43].time := 3600.0, [132].log_data[43].valid := 1, [132].log_data[44].min := -0.30000305, [132].log_data[44].max := -0.27999878, [132].log_data[44].total := -1012.1886, [132].log_data[44].time := 3600.0, [132].log_data[44].minminute := 3, [132].log_data[44].valid := 1, [132].log_data[45].time := 3600.0,
        [132].log_data[45].valid := 1, [132].log_data[46].time := 3600.0, [132].log_data[46].valid := 1, [132].log_data[47].time := 3600.0, [132].log_data[47].valid := 1, [132].log_data[48].min := 6.6673436, [132].log_data[48].max := 6.8066716, [132].log_data[48].total := 24192.055, [132].log_data[48].time := 3600.0, [132].log_data[48].minminute := 27, [132].log_data[48].valid := 1, [132].log_data[49].min := 5.684369, [132].log_data[49].max := 9.011115, [132].log_data[49].total := 25003.557, [132].log_data[49].time := 3600.0, [132].log_data[49].minminute := 20, [132].log_data[49].maxminute := 59, [132].log_data[49].valid := 1, [132].log_data[50].min := 2.00121, [132].log_data[50].max := 2.0113387, [132].log_data[50].total := 7228.0664, [132].log_data[50].time := 3600.0, [132].log_data[50].minminute := 1, [132].log_data[50].maxminute := 58, [132].log_data[50].valid := 1, [132].log_data[51].time := 3600.0, [132].log_data[51].valid := 1, [132].log_data[52].min := -1.6399994, [132].log_data[52].max := -1.4599991, [132].log_data[52].total := -5646.0864, [132].log_data[52].time := 3600.0, [132].log_data[52].minminute := 16, [132].log_data[52].maxminute := 9, [132].log_data[52].valid := 1, [132].log_data[53].min := -1.5800018, [132].log_data[53].max := -1.4000015, [132].log_data[53].total := -5330.179, [132].log_data[53].time := 3600.0, [132].log_data[53].minminute := 38, [132].log_data[53].maxminute := 42, [132].log_data[53].valid := 1, [132].log_data[54].time := 3600.0, [132].log_data[54].valid := 1, [132].log_data[55].time := 3600.0, [132].log_data[55].valid := 1, [132].log_data[56].min := 0.15902862, [132].log_data[56].max := 0.15942119, [132].log_data[56].total := 573.06836, [132].log_data[56].time := 3600.0, [132].log_data[56].minminute := 6, [132].log_data[56].maxminute := 33, [132].log_data[56].valid := 1, [132].log_data[57].min := 0.2009957, [132].log_data[57].max := 0.20138828, [132].log_data[57].total := 724.1395, [132].log_data[57].time := 3600.0, [132].log_data[57].minminute := 31, [132].log_data[57].maxminute := 1, [132].log_data[57].valid := 1, [132].log_data[58].time := 3600.0,
